    # x radius of tri wave
    global x_radius = (move_dis/wv_total_hz)
    # single wave distance
    global wave_dis = sqrt((x_radius*x_radius)+(y_radius*y_radius))*4
    # total robot distance
    global total_dis = wv_total_hz * wave_dis

    # robot speed distance/time = speed
    wv_system_speed = total_dis / (wv_times)
    if(wv_times == 0 or cir_speed_org == 0):
      write_port_register(142,111)
      sleep(0.5)
      halt
    end
    return wv_system_speed
  end


  def set_current_voltage(o_cur,o_vol):
    if(isHicomm):
      set_current_voltage_hicomm(o_cur,o_vol)
    else:
      set_current_voltage_analog(o_cur,o_vol)
    end
  end

  def set_current_voltage_hicomm(o_cur,o_vol):
      write_port_register(204,o_cur)
      write_port_register(205,o_vol*10)
      write_port_register(133,o_cur)
      write_port_register(134,o_vol*10)
  end

  def set_current_voltage_analog(o_cur,o_vol):
      vol_an=((o_vol-14)/2.8)/10
      amp_an=((o_cur-60)/44)/10
      set_standard_analog_out(0,vol_an)
      set_standard_analog_out(1,amp_an)
      write_port_register(133,o_cur)
      write_port_register(134,o_vol*10)
  end

  def calculate_2f(wving_amplitude,tg_wv_wp1,tg_wv_wp2,cir_speed_org,wving_frequency,wving_delay,wving_crater,wving_dir):
    # 진폭
    global y_radius = wving_amplitude / 2
    # 이동 거리
    global move_dis = point_dist(tg_wv_wp1,tg_wv_wp2)*1000
    global move_dis_total = move_dis
    # total running time (sec) - cir_speed_org cpm.
    global wv_times_org = move_dis/(cir_speed_org/6)
    global wv_times = wv_times_org
    global wv_total_hz = floor(wv_times_org*wving_frequency/(1+wving_delay[0]+wving_delay[1]+wving_delay[2]+wving_delay[3]))
    global get_total = wv_total_hz

    dir=1

    ratio_t_sam = 1/get_total
    T1_sam = interpolate_pose(tg_wv_wp1,tg_wv_wp2,ratio_t_sam)
    ratio_t_sam = ratio_t_sam + 1/get_total
    T2_sam = interpolate_pose(tg_wv_wp1,tg_wv_wp2,ratio_t_sam)
    ratio_t_sam = ratio_t_sam + 1/get_total
    T3_sam = interpolate_pose(tg_wv_wp1,tg_wv_wp2,ratio_t_sam)

    push_angle = wving_crater[6]
    push_dis_sam = norm(y_radius)/tan(d2r(push_angle))
    Tp1_sam = feature_offset(T2_sam,p[0,y_radius/1000,0,0,0,0],wv_Line_Feature2)
    Tp2_sam = feature_offset(T2_sam,p[0,-y_radius/1000,0,0,0,0],wv_Line_Feature2)
    Tp1_sam = feature_offset(Tp1_sam,p[wving_dir*push_dis_sam/1000,0,0,0,0,0],wv_Line_Feature2)
    Tp3_sam = feature_offset(T3_sam,p[0,-y_radius/1000,0,0,0,0],wv_Line_Feature2)
    total_step = (get_line_dist(Tp1_sam,Tp2_sam)+get_line_dist(Tp1_sam,Tp3_sam))*1000
    total_dis = wv_total_hz * total_step

    wv_system_speed = (total_dis / wv_times)

    if(wv_times == 0 or cir_speed_org == 0):
      write_port_register(142,111)
      sleep(0.5)
      halt
    end
    return wv_system_speed
  end
  def weaving_simple(wv_wp1,wv_wp3,cir_speed_org,wving_frequency,wving_amplitude,welding_on):
    wv_dist = 0
    tilt_deg = [0,0,0]
    wving_delay = [0,0,0,0]
    wving_type = 1
    Arc_sen=[0,0,0,0,0,0]
    wv_gap=[0,0,0,0]
    welding_dir=1
    z_param=[0,0,0,0,0]
    par_2f=False
    wving_crater=[0,0,0,0,0,0,0,0,0,0]
    ext_fun=[0,0,0,0,0,0,0,0,0,0,0]
    wv_seq = [0,-1]
    wv_feature=p[0,0,0,0,0,0]
    wv_weldpar=[0,cir_speed_org,0,wving_frequency,wving_amplitude,wving_type,welding_dir]
    line_weaving_tp(wv_wp1,wv_wp3,wv_weldpar,tilt_deg,wving_delay,welding_on,Arc_sen,wv_gap,z_param,par_2f,wving_crater,ext_fun,wv_seq,wv_feature)
  end

  def line_weaving_tp(wv_wp1,wv_wp3,wv_weldpar=[100,10,0,1,5,1,1,1,0],tilt_deg=[0,0,0],wving_delay=[0,0,0,0],welding_on=False,Arc_sen=[0,0,0,0,0,0],wv_gap=[0,0,0,0],z_param=[0,0,0,0,0],par_2f=False,wving_crater=[0,0,0,0,0,0,0,0,0,0],ext_fun=[0,0,0,0,0,0,0,0,0,0,0],wv_seq = [0,-1],wv_feature=p[0,0,0,0,0,0]):
    global start_gas_time = 2
    global counter_average = 1
    global counter_average_num = 0
    global waste_cycle = ext_fun[8]
    if(first_half):
      Arc_sen[1] = Arc_sen[1]/2
      Arc_sen[2] = Arc_sen[2]/2
      Arc_sen[3] = Arc_sen[3]/2
      Arc_sen[4] = Arc_sen[4]/2
    end
    global arc_x_off=0
    global arc_z_off=0
    global Up = 0
    global Ui = 0
    global Up_z = 0
    global Ui_z = 0
    if(wv_weldpar[7] == 1):
      global record_multi = False
    else:
      global record_multi = True
    end
    global th_ext_fun = ext_fun
    RTDE_init()

    # e-Series 2, CB-Seris 8
    global system_bus_ms = 2

    global sin_dir = wv_seq[1]
    global start_trig = False
    dir=1
    if(par_2f):
      global squash_cycle = 0
      # sin_dir = sin_dir
      sin_dir = sin_dir * -1
    else:
      global squash_cycle = ext_fun[7]
    end
    global tri_count=0

    global z_bottom = z_param[0]/1000
    if(wv_weldpar[6]==-1):
      #right
      global vir_v = -1
    else:
      #left
      global vir_v = 1
    end

    if(par_2f):
      global cal_off_ang_rx = 1
      global cal_off_ang_ry = 0
    else:
      global cal_off_ang_rx = 0
      global cal_off_ang_ry = 1
    end

    if(wv_seq[0] == 2 or wv_seq[0] == 3):
      tilt_deg = [0,0,0]
      global cal_off_ang_rx = 0
      global cal_off_ang_ry = 0
    end

    global wv_Line_Feature2 = wv_wp1
    if(wv_weldpar[0] > 650 and par_2f == False):
      wv_weldpar[0] = 650
    end
    if(wv_wp3==p[0,0,0,0,0,0]):
      global wv_wp2 = feature_offset(wv_wp1,p[wv_weldpar[0]/1000,0,0,0,0,0],wv_Line_Feature2)
    else:
      global wv_wp2 = wv_wp3
      wv_weldpar[0] = point_dist(wv_wp1,wv_wp2)*1000
      global wv_dist_bak = point_dist(wv_wp1,wv_wp2)*1000
    end
    if(wv_feature != p[0,0,0,0,0,0]):
      wv_Line_Feature2 = wv_feature
    end
    if(vir_v==1):
      line_x = get_feature_Line(wv_wp1,wv_wp2)
    else:
      line_x = get_feature_Line(wv_wp2,wv_wp1)
    end
    pp1 = feature_offset(wv_wp1,p[0,20/1000,0,0,0,0],line_x)
    pp2 = pose_add(wv_wp1,p[0,0,20/1000,0,0,0])
    global wp_Feature = get_feature_plane_yz(wv_wp1,pp1,pp2)

    #setting
    if(par_2f):
      #todo - 1
      global offset_2f_k = -1 * ext_fun[9]
      global offset_2f_z = 1 * ext_fun[10]
      if(wv_seq[0] == 0 or wv_seq[0] == 1):
        # line_feature = get_feature_Line(wv_wp1,wv_wp2)
        line_feature = get_feature_Line(wv_wp2,wv_wp1)
        b_p1 = wv_wp1
        b_p2 = feature_offset(wv_wp1,p[0,0.02*vir_v,0,0,0,0],line_feature)
        # b_p2 = feature_offset(wv_wp1,p[0,0.01,0,0,0,0],line_feature)
        b_p3 = pose_add(wv_wp1,p[0,0,0.02,0,0,0])

        global back_feature = get_feature_plane_xz(b_p1,b_p2,b_p3)

        wv_wp1 = pose_trans(wv_wp1,p[0,0,0,0,0,d2r(-90)])
        wv_wp1 = feature_offset(wv_wp1,p[0,offset_2f_k/1000,0,0,0,0],back_feature)
        wv_wp1 = pose_add(wv_wp1,p[0,0,offset_2f_z/1000,0,0,0])
        global bak_wv_wp1 = wv_wp1
      end
        wv_wp2 = feature_offset(wv_wp2,p[0,offset_2f_k/1000,0,0,0,0],back_feature)
        wv_wp2 = pose_add(wv_wp2,p[0,0,offset_2f_z/1000,0,0,0])
        wv_wp2 = p[wv_wp2[0],wv_wp2[1],wv_wp2[2],wv_wp1[3],wv_wp1[4],wv_wp1[5]]
        global bak_wv_wp2 = wv_wp2
    end
    if(ext_fun[2]==1 and par_2f==False):
      w_voltage = ext_fun[3]
      w_current = ext_fun[4]
      set_current_voltage(w_current,w_voltage)
      global cir_speed_org_bak = wv_weldpar[1]
      global wving_amplitude_bak = wv_weldpar[4]
      wv_weldpar[1] = ext_fun[6]
      wv_weldpar[4] = ext_fun[5]
    end
    if(par_2f):
      global wv_system_speed = calculate_2f(wv_weldpar[4],wv_wp1,wv_wp2,wv_weldpar[1],wv_weldpar[3],wving_delay,wving_crater,wv_weldpar[6])
    else:
      global wv_system_speed = calculate_3f(wv_weldpar[4],wv_wp1,wv_wp2,wv_weldpar[1],wv_weldpar[3],wving_delay)
      x_radius = x_radius / 1000
    end
    global wv_set_speed = wv_system_speed
    ratio_t=0
    global y_radius = y_radius / 1000
    global y_radius_bak = y_radius
    global ext_stick = 0
    global th_arc_sen=Arc_sen
    global th_wv_gap=wv_gap
    global th_tilt_deg=tilt_deg
    global last_tilt_deg = th_tilt_deg
    global last_wv_wp1 = wv_wp1
    global last_wv_line = wv_Line_Feature2
    global last_z_bottom = z_bottom
    global th_wving_crater=wving_crater
    global th_par_2f = par_2f
    global th_cir_speed_org=wv_weldpar[1]
    global th_wv_wp1 = wv_wp1
    global th_wv_wp2 = wv_wp2
    global th_wv_wp3 = wv_wp3
    global th_wv_weldpar=wv_weldpar
    global th_wving_delay=wving_delay
    global th_z_param=z_param
    global th_wv_seq = wv_seq
    global th_wv_feature=wv_feature
    global th_dir = dir

    # if want to use approach position
    if(wv_seq[0] ==0 or wv_seq[0] == 1):
      global get_angle_rx = welding_angle_cal_2f(wv_wp1[1],tilt_deg,vir_v,cal_off_ang_rx)
      global get_angle_ry = welding_angle_cal_3f(wv_wp1[2],tilt_deg,z_bottom,cal_off_ang_ry)

      target_p = feature_offset(wv_wp1,p[0,0,0,d2r(tilt_deg[0] + get_angle_rx),d2r(tilt_deg[1] + get_angle_ry),d2r(tilt_deg[2])],wv_Line_Feature2)

      if(wv_weldpar[2]==1):
        target_p_appr = feature_offset(target_p,p[0,0,-0.02,0,0,0],wv_Line_Feature2)
        movel(target_p_appr,a=0.5,v=0.125)
      end
      movel(target_p,a=0.5,v=0.125)
    end
    CThread = run CalThread()
    DThread = run diff_Thread()
    TThread = run thread_timer()
    AThread = run Arc_Thread()
    TTRRhread = run thread_dist_rec()

    global timer_counting=True
    global program_weld_on = True

    if(a9_wv_weldingon==True):
      while(welding_off_t==55):
        sync()
      end
      if(wving_crater[2]>0):
        set_current_voltage(wving_crater[0],wving_crater[1])
      end
      if(welding_off_t != 1):
        if(isHicomm):
          write_welder(0,True)
        else:
          set_standard_digital_out(0,True)
        end
        while(read_welder(5)==False):
          if(weld_onoff==False):
              write_welder(0,True)
          end
          sync()
        end
        if(wving_crater[2]>0):
          #Crater Begin option
          write_output_float_register(1,1)
          sleep(wving_crater[2])
          set_current_voltage(ext_fun[1],ext_fun[0])
        end
      end
    end
    start_gas_time = 0

    background_cal=1
    background_ready=0
    FT_trig=True
    timer_1_is_counting = True
    global welding_program = False

    while((ratio_t < 1)):
      if( (norm(tri_count)>=2 and par_2f==False or FT_trig==True) or (norm(tri_count)>=4 and par_2f or FT_trig==True) ):
        FT_trig = False
        while(background_ready==0):
          sync()
        end
        tri_count = 0
        background_ready = 0
        global move_p = background_pose
        wv_wp2 = th_wv_wp2
        if(par_2f):
          background_cal=1
        else:
          background_cal=1
        end
        global a_val = 3
        if(a_val >= 30):
          write_port_register(142,112)
          sleep(0.5)
          halt
        end
      end
      if(wv_weldpar[5] ==1):
          if( (sin_dir==1 and wving_delay[0]==0) or (sin_dir==-1 and wving_delay[2]==0)):
           tri_count = tri_count + 1
          end
          global target_p = move_p[tri_count]
          # write_output_float_register(24,tri_count)
          # target_p=p[target_p[0],target_p[1],target_p[2],target_p[3],target_p[4],target_p[5]]
          tri_count = tri_count + 1
      elif(wv_weldpar[5] ==2):
        if((tri_count==0 and wving_delay[2]==0) or (tri_count==2 and wving_delay[0]==0)):
         tri_count = tri_count + 1
        end
        global target_p = move_p[tri_count]
        # write_output_float_register(24,tri_count)
        # target_p=p[target_p[0],target_p[1],target_p[2],target_p[3],target_p[4],target_p[5]]
        tri_count = tri_count + 1
      else:
        popup("Please insert 0 - sin or 1 - triangle")
      end
      if(target_p == p[0,0,0,0,0,0]):
        target_p = get_actual_tcp_pose()
      end
      #3F tri_count 2 는 tri_count가 계속 move_p[1]만 간다

      # write_output_float_register(23,sin_dir)

      ARC_T_ONOFF = True
      ARC_T_s_pose = get_actual_tcp_pose()
      ARC_T_e_pose = target_p
      if((norm(tri_count)== 2) and wving_delay[1]>0 and par_2f):
        #down
        movel(target_p,a=a_val,v=wv_system_speed/1000)
        sleep(wving_delay[1])
      elif((norm(tri_count)== 4) and wving_delay[3]>0 and par_2f):
        #4
        movel(target_p,a=a_val,v=wv_system_speed/1000)
        sleep(wving_delay[3])
      elif((norm(tri_count)== 2) and sin_dir==1 and wving_delay[1]>0 and par_2f == False):
        movel(target_p,a=a_val,v=wv_system_speed/1000)
        sleep(wving_delay[1])
      elif((norm(tri_count)== 2) and sin_dir==-1 and wving_delay[3]>0 and par_2f == False):
        movel(target_p,a=a_val,v=wv_system_speed/1000)
        sleep(wving_delay[3])
      elif((norm(tri_count)== 1) and wving_delay[2]>0 and par_2f):
        movel(target_p,a=a_val,v=wv_system_speed/1000)
        sleep(wving_delay[2])
      elif((norm(tri_count)== 3) and wving_delay[0]>0 and par_2f):
        #3
        movel(target_p,a=a_val,v=wv_system_speed/1000)
        sleep(wving_delay[0])
      else:
        movel(target_p,a=a_val,v=wv_system_speed/1000)
      end
      global last_pose = target_p
    end
    timer_1_is_counting = False

    if(a9_wv_weldingon == True and wving_crater[5]!=0):
      #crater end option
      set_current_voltage(wving_crater[3],wving_crater[4])
      sleep(wving_crater[5])
      program_weld_on = False
      set_current_voltage(ext_fun[1],ext_fun[0])
      if(isHicomm):
        write_port_register(202,0)
        write_port_register(149,0)
      else:
        set_standard_digital_out(0,False)
      end
      while(read_welder(5)==True):
        if(weld_onoff==True):
          write_welder(0,False)
        end
        sync()
      end
    end
    timer_counter = 0
    kill CThread
    kill DThread
    kill TThread
    kill AThread
    kill TTRRhread
    ARC_T_ONOFF=False
    timer_counter = 0
    timer_counting = False
    wcr_counter = 0
    wcr_counting = False
    get_wcr = False
    welding_off_t = 0
    plus_alpha_x = 0
    plus_alpha_z = 0

    if(wv_seq[0] == 0 or wv_seq[0] == 3):
      if(a9_wv_weldingon==True):
        program_weld_on = False
        write_port_register(202,0)
        write_port_register(149,0)
        write_welder(0,False)
        if(wv_weldpar[2]==1):
          target_pos = feature_offset(get_actual_tcp_pose(),p[0,0,-0.01,0,0,0],wv_Line_Feature2)
          movel(target_pos,0.5,0.01)
        end
      end
    end
    background_pose = [dumy_p,dumy_p,dumy_p,dumy_p]
    move_p = background_pose
    return sin_dir
  end


  def line_weaving_tp_l(wv_wp1,wv_wp3,wv_weldpar=[100,10,0,1,5,1,1,1,0],tilt_deg=[0,0,0],wving_delay=[0,0,0,0],welding_on=False,Arc_sen=[0,0,0,0,0,0],wv_gap=[0,0,0,0],z_param=[0,0,0,0,0],par_2f=False,wving_crater=[0,0,0,0,0,0,0,0,0,0],ext_fun=[0,0,0,0,0,0,0,0,0,0,0],wv_seq = [0,-1],wv_feature=p[0,0,0,0,0,0]):
    global start_gas_time = 2
    global counter_average = 1
    global counter_average_num = 0
    global waste_cycle = ext_fun[8]
    if(first_half):
      Arc_sen[1] = Arc_sen[1]/2
      Arc_sen[2] = Arc_sen[2]/2
      Arc_sen[3] = Arc_sen[3]/2
      Arc_sen[4] = Arc_sen[4]/2
    end
    global current_list = 0
    global wv_wp4 = wv_wp3
    global A_T1 = wv_wp4[0]
    global A_T2 = wv_wp4[1]
    global A_T3 = wv_wp4[2]

    global arc_x_off=0
    global arc_z_off=0
    global Up = 0
    global Ui = 0
    global Up_z = 0
    global Ui_z = 0
    global th_ext_fun = ext_fun
    if(wv_weldpar[7] == 1):
      global record_multi = False
    else:
      global record_multi = True
    end
    RTDE_init()

    if (wv_gap[0]==1):
      gap_check = True
      wv_gap[0]=0
    else:
      gap_check= False
    end
    # e-Series 2, CB-Seris 8
    global system_bus_ms = 2

    global sin_dir = wv_seq[1]
    if(par_2f):
      global squash_cycle = 0
      # sin_dir = sin_dir
      sin_dir = sin_dir * -1
    else:
      global squash_cycle = ext_fun[7]
    end
    global start_trig = False
    dir=1

    global tri_count=0

    global z_bottom = z_param[0]/1000
    if(wv_weldpar[6]==-1):
      global vir_v = -1
    else:
      global vir_v = 1
    end

    if(par_2f):
      global cal_off_ang_rx = 1
      global cal_off_ang_ry = 0
    else:
      global cal_off_ang_rx = 0
      global cal_off_ang_ry = 1
    end

    if(wv_seq[0] == 2 or wv_seq[0] == 3):
      tilt_deg = [0,0,0]
      global cal_off_ang_rx = 0
      global cal_off_ang_ry = 0
    end

    global wv_Line_Feature2 = wv_wp1
    if(wv_weldpar[0] > 700 and par_2f == False):
      wv_weldpar[0] = 700
    end
    if(wv_wp3[0]==p[0,0,0,0,0,0]):
      global wv_wp2 = feature_offset(wv_wp1,p[wv_weldpar[0]/1000,0,0,0,0,0],wv_Line_Feature2)
    else:
      global wv_wp2 = wv_wp4[0]
      wv_weldpar[0] = point_dist(wv_wp1,wv_wp2)*1000
      global wv_dist_bak = point_dist(wv_wp1,wv_wp2)*1000
    end
    if(wv_seq[0] == 2 or wv_seq[0] == 3):
      wv_Line_Feature2 = wv_feature
    end
    if(vir_v==1):
      line_x = get_feature_Line(wv_wp1,wv_wp2)
    else:
      line_x = get_feature_Line(wv_wp2,wv_wp1)
    end  pp1 = feature_offset(wv_wp1,p[0,20/1000,0,0,0,0],line_x)
    pp2 = pose_add(wv_wp1,p[0,0,20/1000,0,0,0])
    global wp_Feature = get_feature_plane_yz(wv_wp1,pp1,pp2)

    #setting
    if(par_2f):
      #todo - 1
      offset_2f_k = -1 * ext_fun[9]
      offset_2f_z = 1 * ext_fun[10]
      if(wv_seq[0] == 0 or wv_seq[0] == 1):
        line_feature = get_feature_Line(wv_wp1,wv_wp2)
        b_p1 = wv_wp1
        b_p2 = feature_offset(wv_wp1,p[0,0.01*vir_v,0,0,0,0],line_feature)
        b_p3 = pose_add(wv_wp1,p[0,0,0.01,0,0,0])

        back_feature = get_feature_plane_xz(b_p1,b_p2,b_p3)
        wv_wp1 = pose_trans(wv_wp1,p[0,0,0,0,0,d2r(-90)])
        wv_wp1 = feature_offset(wv_wp1,p[0,offset_2f_k/1000,0,0,0,0],back_feature)
        wv_wp1 = pose_add(wv_wp1,p[0,0,offset_2f_z/1000,0,0,0])
        # wv_wp1 = pose_add(wv_wp1,p[offset_2f_k/1000,0,0,0,0,0])
      end
        # wv_wp2 = pose_add(wv_wp2,p[offset_2f_k/1000,0,0,0,0,0])
        wv_wp2 = feature_offset(wv_wp2,p[0,offset_2f_k/1000,0,0,0,0],back_feature)
        wv_wp2 = pose_add(wv_wp2,p[0,0,offset_2f_z/1000,0,0,0])
        wv_wp2 = p[wv_wp2[0],wv_wp2[1],wv_wp2[2],wv_wp1[3],wv_wp1[4],wv_wp1[5]]

        wv_wp3_p = feature_offset(wv_wp3[0],p[0,offset_2f_k/1000,0,0,0,0],back_feature)
        wv_wp3_p = pose_add(wv_wp3_p,p[0,0,offset_2f_z/1000,0,0,0])
        wv_wp3_p = p[wv_wp3_p[0],wv_wp3_p[1],wv_wp3_p[2],wv_wp1[3],wv_wp1[4],wv_wp1[5]]
        wv_wp4[0] = p[wv_wp3_p[0],wv_wp3_p[1],wv_wp3_p[2],wv_wp1[3],wv_wp1[4],wv_wp1[5]]

        wv_wp3_p = feature_offset(wv_wp3[1],p[0,offset_2f_k/1000,0,0,0,0],back_feature)
        wv_wp3_p = pose_add(wv_wp3_p,p[0,0,offset_2f_z/1000,0,0,0])
        wv_wp3_p = p[wv_wp3_p[0],wv_wp3_p[1],wv_wp3_p[2],wv_wp1[3],wv_wp1[4],wv_wp1[5]]
        wv_wp4[1] = p[wv_wp3_p[0],wv_wp3_p[1],wv_wp3_p[2],wv_wp1[3],wv_wp1[4],wv_wp1[5]]

        wv_wp3_p = feature_offset(wv_wp3[2],p[0,offset_2f_k/1000,0,0,0,0],back_feature)
        wv_wp3_p = pose_add(wv_wp3_p,p[0,0,offset_2f_z/1000,0,0,0])
        wv_wp3_p = p[wv_wp3_p[0],wv_wp3_p[1],wv_wp3_p[2],wv_wp1[3],wv_wp1[4],wv_wp1[5]]
        wv_wp4[2] = p[wv_wp3_p[0],wv_wp3_p[1],wv_wp3_p[2],wv_wp1[3],wv_wp1[4],wv_wp1[5]]
    end
    if(ext_fun[2]==1 and par_2f==False):
      #squash
      w_voltage = ext_fun[3]
      w_current = ext_fun[4]
      set_current_voltage(w_current,w_voltage)
      global cir_speed_org_bak = wv_weldpar[1]
      global wving_amplitude_bak = wv_weldpar[4]
      wv_weldpar[1] = ext_fun[6]
      wv_weldpar[4] = ext_fun[5]
    end
    if(par_2f):
      global wv_system_speed = calculate_2f(wv_weldpar[4],wv_wp1,wv_wp2,wv_weldpar[1],wv_weldpar[3],wving_delay,wving_crater,wv_weldpar[6])
    else:
      global wv_system_speed = calculate_3f(wv_weldpar[4],wv_wp1,wv_wp2,wv_weldpar[1],wv_weldpar[3],wving_delay)
      x_radius = x_radius / 1000
    end
    global wv_set_speed = wv_system_speed
    ratio_t=0
    # mm -> m
    global y_radius = y_radius / 1000
    global y_radius_bak = y_radius
    #init for thread
    global ext_stick = 0
    global th_arc_sen=Arc_sen
    global th_wv_gap=wv_gap
    global th_tilt_deg=tilt_deg

    global last_tilt_deg =th_tilt_deg
    global last_wv_wp1 = wv_wp1
    global last_wv_line = wv_Line_Feature2
    global th_wving_crater=wving_crater
    global last_z_bottom = z_bottom
    global th_par_2f = par_2f
    global th_cir_speed_org=wv_weldpar[1]
    global th_wv_wp1 = wv_wp1
    global th_wv_wp2 = wv_wp2
    global th_wv_wp3 = wv_wp3[0]
    global th_wv_weldpar=wv_weldpar
    global th_wving_delay=wving_delay
    global th_z_param=z_param
    global th_wv_seq = wv_seq
    global th_wv_feature=wv_feature
    global th_dir = dir

    # if want to use approach position
    if(wv_seq[0] ==0 or wv_seq[0] == 1):
      global get_angle_rx = welding_angle_cal_2f(wv_wp1[1],tilt_deg,vir_v,cal_off_ang_rx)
      global get_angle_ry = welding_angle_cal_3f(wv_wp1[2],tilt_deg,z_bottom,cal_off_ang_ry)

      target_p = feature_offset(wv_wp1,p[0,0,0,d2r(tilt_deg[0] + get_angle_rx),d2r(tilt_deg[1] + get_angle_ry),d2r(tilt_deg[2])],wv_Line_Feature2)

      if(wv_weldpar[2]==1):
        target_p_appr = feature_offset(target_p,p[0,0,-0.02,0,0,0],wv_Line_Feature2)
        movel(target_p_appr,a=0.5,v=0.125)
      end
      movel(target_p,a=0.5,v=0.125)
    end

    CThread = run CalThread()
    DThread = run diff_Thread()
    TThread = run thread_timer()
    AThread = run Arc_Thread()
    TTRRhread = run thread_dist_rec()

    global timer_counting=True
    global program_weld_on = True

    if(a9_wv_weldingon==True):
      while(welding_off_t==55):
        sync()
      end
      if(wving_crater[2]>0):
        set_current_voltage(wving_crater[0],wving_crater[1])
      end
      if(welding_off_t != 1):
        write_welder(0,True)
        while(get_wcr==False):
          if(weld_onoff==False):
            write_welder(0,True)
          end
          sync()
        end
        if(wving_crater[2]>0):
          #Crater Begin option
          write_output_float_register(1,1)
          sleep(wving_crater[2])
          set_current_voltage(ext_fun[1],ext_fun[0])
        end
      end
    end
    start_gas_time = 0

    background_cal=1
    background_ready=0
    FT_trig=True

    timer_1_is_counting = True

    while((ratio_t < 1) or current_list==0 or current_list==1):
      if(ratio_t>=1 and current_list!=2):
        if (gap_check):
          gap_check = True
          wv_gap[0]=1
          th_wv_gap[0]=1
          gap_check= False
        end
        ratio_t=0
        if(current_list==0):
          wving_amp_bak = wv_weldpar[4]
          wv_weldpar[4] = wv_weldpar[4] * 1
          th_wv_weldpar[4] = wv_weldpar[4]
          circle_speed_bak = wv_weldpar[1]
          wv_weldpar[1]= wv_weldpar[1]*0.7
          th_wv_weldpar[1]= wv_weldpar[1]
        elif(current_list==1):
          wv_weldpar[4] = wving_amp_bak
          th_wv_weldpar[4] = wv_weldpar[4]
          wv_weldpar[1] = circle_speed_bak
          th_wv_weldpar[1]= wv_weldpar[1]
        end
        wv_wp1=wv_wp4[current_list]
        wv_wp2=wv_wp4[current_list+1]
        global th_wv_wp1 = wv_wp4[current_list]
        global th_wv_wp2 = wv_wp4[current_list+1]
        global th_wv_wp3 = wv_wp4[current_list+1]
        wv_system_speed_bak = wv_system_speed
        if(par_2f):
          global wv_system_speed = calculate_2f(wv_weldpar[4],wv_wp4[current_list],wv_wp4[current_list+1],wv_weldpar[1],wv_weldpar[3],wving_delay,wving_crater)
          global y_radius = y_radius / 1000
          global y_radius_bak = y_radius
        else:
          global wv_system_speed = calculate_3f(wv_weldpar[4],wv_wp4[current_list],wv_wp4[current_list+1],wv_weldpar[1],wv_weldpar[3],wving_delay)
          x_radius = x_radius / 1000
        end
        wv_system_speed = wv_system_speed_bak
        current_list=current_list+1
      end

      if( (norm(tri_count)>=2 and par_2f==False or FT_trig==True) or (norm(tri_count)>=4 and par_2f==True or FT_trig==True)   ):
        FT_trig = False
        while(background_ready==0):
          sync()
        end
        tri_count = 0
        background_ready = 0
        global move_p = background_pose
        wv_wp2 = th_wv_wp2
        if(par_2f):
          background_cal=1
        else:
          background_cal=1
        end
        global a_val = 3
        if(a_val >= 30):
          write_port_register(142,112)
          sleep(0.5)
          halt
        end
      end

      if(wv_weldpar[5] ==1):
          if( (sin_dir==1 and wving_delay[0]==0) or (sin_dir==-1 and wving_delay[2]==0)):
           tri_count = tri_count + 1
          end
          # write_output_float_register(24,tri_count)
          global target_p = move_p[tri_count]
          target_p=p[target_p[0],target_p[1],target_p[2],target_p[3],target_p[4],target_p[5]]
          tri_count = tri_count + 1
      elif(wv_weldpar[5] ==2):
        if( (tri_count==1 and sin_dir==1 and wving_delay[0]==0) or (tri_count==1 and sin_dir==-1 and wving_delay[2]==0)):
         tri_count = tri_count + 1
        end
        # write_output_float_register(24,tri_count)
        global target_p = move_p[tri_count]
        target_p=p[target_p[0],target_p[1],target_p[2],target_p[3],target_p[4],target_p[5]]
        tri_count = tri_count + 1
      else:
        popup("Please insert 0 - sin or 1 - triangle")
      end

      if(target_p == p[0,0,0,0,0,0]):
        target_p = get_actual_tcp_pose()
      end
      # write_output_float_register(23,sin_dir)
      ARC_T_ONOFF = True
      ARC_T_s_pose = get_actual_tcp_pose()
      ARC_T_e_pose = target_p
      if((norm(tri_count)== 2) and wving_delay[1]>0 and par_2f):
        # DOWN
        movel(target_p,a=a_val,v=wv_system_speed/1000)
        sleep(wving_delay[1])
      elif((norm(tri_count)== 4) and wving_delay[3]>0 and par_2f):
        #UP
        movel(target_p,a=a_val,v=wv_system_speed/1000)
        sleep(wving_delay[3])
      elif((norm(tri_count)== 2) and sin_dir==1 and wving_delay[1]>0 and par_2f == False):
        movel(target_p,a=a_val,v=wv_system_speed/1000)
        sleep(wving_delay[1])
      elif((norm(tri_count)== 2) and sin_dir==-1 and wving_delay[3]>0 and par_2f == False):
        movel(target_p,a=a_val,v=wv_system_speed/1000)
        sleep(wving_delay[3])
      elif((norm(tri_count)== 1) and wving_delay[0]>0 and par_2f):
        movel(target_p,a=a_val,v=wv_system_speed/1000)
        sleep(wving_delay[0])
      elif((norm(tri_count)== 3) and wving_delay[2]>0 and par_2f):
        movel(target_p,a=a_val,v=wv_system_speed/1000)
        sleep(wving_delay[2])
      else:
        movel(target_p,a=a_val,v=wv_system_speed/1000)
      end
      global last_pose = target_p
    end

    timer_1_is_counting = False
    welding_program = True
    if(a9_wv_weldingon == True and wving_crater[5]!=0):
      #crater end option
      set_current_voltage(wving_crater[3],wving_crater[4])
      sleep(wving_crater[5])
      program_weld_on = False
      set_current_voltage(ext_fun[1],ext_fun[0])
      if(isHicomm):
        write_port_register(202,0)
        write_port_register(149,0)
      else:
        set_standard_digital_out(0,False)
      end
      while(get_wcr==True):
        if(weld_onoff==True):
          if(isHicomm):
            write_port_register(202,0)
            write_port_register(149,0)
          else:
            set_standard_digital_out(0,False)
          end
        end
        sync()
      end
    end

    kill CThread
    kill DThread
    kill TThread
    kill AThread
    kill TTRRhread
    ARC_T_ONOFF=False
    timer_counting = False
    wcr_counter = 0
    wcr_counting = False
    get_wcr = False
    welding_off_t = 0
    plus_alpha_x = 0
    plus_alpha_z = 0

    if(wv_seq[0] == 0 or wv_seq[0] == 3):
      if(a9_wv_weldingon==True):
        program_weld_on = False
        if(isHicomm):
          write_port_register(202,0)
          write_port_register(149,0)
        else:
          set_standard_digital_out(0,False)
        end
        if(wv_weldpar[2]==1):
          target_pos = feature_offset(get_actual_tcp_pose(),p[0,0,-0.01,0,0,0],wv_Line_Feature2)
          movel(target_pos,0.5,0.01)
        end
      end
    end
    background_pose = [dumy_p,dumy_p,dumy_p,dumy_p]
    move_p = background_pose
    return sin_dir
  end
  $ 152 "Reset"
  $ 153 "If Reset_Trig"
  if (Reset_Trig):
    $ 154 "Reset_Trig≔ False "
    global Reset_Trig=  False
    $ 155 "Call robotand_cell_initalizat"
    robotand_cell_initalizat()
    $ 156 "Auto_trig≔ False "
    global Auto_trig=  False
    $ 157 "write_port_register(cell_3f_2f_151,0)"
    write_port_register(cell_3f_2f_151,0)
    $ 158 "write_port_register(cell_info_152,0)"
    write_port_register(cell_info_152,0)
    $ 159 "write_port_register(weld_req_153,0)"
    write_port_register(weld_req_153,0)
    $ 160 "write_port_register(return_done_240,0)"
    write_port_register(return_done_240,0)
    $ 161 "write_port_register(robot_move_163,0)"
    write_port_register(robot_move_163,0)
    $ 162 "write_port_register(robot_pose_164,0)"
    write_port_register(robot_pose_164,0)
    $ 163 "write_port_register(182,0)"
    write_port_register(182,0)
    $ 164 "write_port_register(185,0)"
    write_port_register(185,0)
    $ 165 "write_port_register(201,0)"
    write_port_register(201,0)
    $ 166 "write_port_register(202,0)"
    write_port_register(202,0)
  end
  $ 167 "Welding_Init"
  $ 168 "'welding parameter initialization'"
  # 'welding parameter initialization'
  $ 169 "welding_etc"
  $ 197 "c5_wv_gap_y≔0"
  global c5_wv_gap_y=0
  $ 198 "c6_wv_gap_cpm≔0"
  global c6_wv_gap_cpm=0
  $ 199 "c9_wv_gap_freq≔0"
  global c9_wv_gap_freq=0
  $ 200 "c4_gap_enable≔0"
  global c4_gap_enable=0
  $ 201 "c7_wv_gap≔[c4_gap_enable,c5_wv_gap_y,c6_wv_gap_cpm,c9_wv_gap_freq]"
  global c7_wv_gap=[c4_gap_enable,c5_wv_gap_y,c6_wv_gap_cpm,c9_wv_gap_freq]
  $ 202 "init_reset_modbus_server"
  $ 203 "set_tool_voltage(24)"
  set_tool_voltage(24)
  $ 204 "write_port_register(163,0)"
  write_port_register(163,0)
  $ 205 "write_port_register(164,0)"
  write_port_register(164,0)
  $ 207 "write_port_register(201,1)"
  write_port_register(201,1)
  $ 208 "write_port_register(202,0)"
  write_port_register(202,0)
  $ 1310 "Thread_2"
  thread Thread_2():
    while (True):
      $ 1311 "Thread_heartbeat"
      $ 1312 "heartbeat≔heartbeat+1"
      global heartbeat=heartbeat+1
      $ 1313 "If heartbeat>499"
      if (heartbeat>499):
        $ 1314 "heartbeat≔0"
        global heartbeat=0
      end
      $ 1315 "write_port_register(128,heartbeat)"
      write_port_register(128,heartbeat)
      $ 1325 "Wait: 1.0"
      sleep(1.0)
    end
  end
  threadId_Thread_2 = run Thread_2()
  $ 1326 "Thread_1"
  thread Thread_1():
    while (True):
      $ 1327 "thread main"
      $ 1328 "a0_Job_Mode≔read_port_register(162)"
      global a0_Job_Mode= read_port_register (162)
      $ 1329 "a1_job_move≔read_port_register(163)"
      global a1_job_move= read_port_register (163)
      $ 1330 "If red_led≟ True "
      if (get_tool_digital_out(0) ==   True  ):
        $ 1331 "Set red_led=Off"
        set_tool_digital_out(0, False)
      end
      $ 1332 "If a0_Job_Mode≟2"
      if (a0_Job_Mode == 2):
        $ 1333 "If read_port_register(arc_onoff_168)≟2"
        if ( read_port_register (arc_onoff_168) == 2):
          $ 1334 "a9_wv_weldingon≔ True "
          global a9_wv_weldingon=  True
        else:
          $ 1335 "Else" "noBreak"
          $ 1336 "a9_wv_weldingon≔ False "
          global a9_wv_weldingon=  False
        end
        $ 1337 "If Auto_trig"
        if (Auto_trig):
          $ 1338 "get_next_number≔read_port_register(166)"
          global get_next_number= read_port_register (166)
          $ 1339 "get_move_trig≔read_port_register(167)"
          global get_move_trig= read_port_register (167)
          $ 1340 "If get_move_trig≟1 and running_trig≟ True "
          if (get_move_trig == 1  and  running_trig ==   True  ):
            $ 1341 "If get_next_number<0 or get_next_number>30"
            if (get_next_number<0  or  get_next_number>30):
              $ 1342 "write_port_register(142,141)"
              write_port_register(142,141)
              $ 1343 "Halt"
              halt
            end
            $ 1344 "If get_next_number≠Auto_cur_cell"
            if (get_next_number != Auto_cur_cell):
              $ 1345 "running_trig≔ False "
              global running_trig=  False
              $ 1346 "write_welder(0, False )"
              write_welder(0,  False  )
              $ 1347 "write_port_register(149,0)"
              write_port_register(149,0)
              $ 1348 "write_port_register(202,0)"
              write_port_register(202,0)
            else:
              $ 1349 "Else" "noBreak"
              $ 1350 "write_port_register(166,0)"
              write_port_register(166,0)
              $ 1351 "write_port_register(167,0)"
              write_port_register(167,0)
            end
          end
        end
        $ 1352 "If t_time>timer_1"
        if (t_time>timer_1):
          $ 1353 "write_port_register(143,timer_1)"
          write_port_register(143,timer_1)
        else:
          $ 1354 "Else" "noBreak"
          $ 1355 "write_port_register(143,timer_1)"
          write_port_register(143,timer_1)
          $ 1356 "write_port_register(144,timer_1)"
          write_port_register(144,timer_1)
        end
        $ 1357 "Monitoring touch and welding"
        $ 1358 "If read_welder_control(0) and read_port_register(130)≠1"
        if (read_welder_control(0)  and   read_port_register (130) != 1):
          $ 1359 "write_port_register(130,1)"
          write_port_register(130,1)
        else:
          $ 1360 "ElseIf read_welder_control(0) and read_port_register(130)≠0"
          if (read_welder_control(0)  and   read_port_register (130) != 0):
            $ 1361 "write_port_register(130,0)"
            write_port_register(130,0)
          end
        end
        $ 1362 "If read_welder(5)"
        if (read_welder(5)):
          $ 1363 "'check wcr in (digital)'"
          # 'check wcr in (digital)'
          $ 1364 "write_output_float_register(20,1)"
          write_output_float_register(20,1)
        else:
          $ 1365 "Else" "noBreak"
          $ 1366 "write_output_float_register(20,0)"
          write_output_float_register(20,0)
        end
        $ 1367 "If read_welder(4)"
        if (read_welder(4)):
          $ 1368 "'check touch (digital)'"
          # 'check touch (digital)'
          $ 1369 "write_output_float_register(21,1)"
          write_output_float_register(21,1)
        else:
          $ 1370 "Else" "noBreak"
          $ 1371 "write_output_float_register(21,0)"
          write_output_float_register(21,0)
        end
        $ 1372 "If read_welder_control(0)"
        if (read_welder_control(0)):
          $ 1373 "'check welding out (digital)'"
          # 'check welding out (digital)'
          $ 1374 "write_output_float_register(17,1)"
          write_output_float_register(17,1)
        else:
          $ 1375 "Else" "noBreak"
          $ 1376 "write_output_float_register(17,0)"
          write_output_float_register(17,0)
        end
        $ 1377 "If read_welder_control(4)"
        if (read_welder_control(4)):
          $ 1378 "'check touch out (digital)'"
          # 'check touch out (digital)'
          $ 1379 "write_output_float_register(18,1)"
          write_output_float_register(18,1)
        else:
          $ 1380 "Else" "noBreak"
          $ 1381 "write_output_float_register(18,0)"
          write_output_float_register(18,0)
        end
      end
      $ 1382 "If get_tool_digital_in(1)≟ True "
      if (get_tool_digital_in(1) ==   True  ):
        $ 1383 "set_tool_digital_out(1, False )"
        set_tool_digital_out(1,  False  )
      else:
        $ 1384 "Else" "noBreak"
        $ 1385 "set_tool_digital_out(1, True )"
        set_tool_digital_out(1,  True  )
      end
      $ 1386 "If red_led≟ True "
      if (get_tool_digital_out(0) ==   True  ):
        $ 1387 "Set red_led=Off"
        set_tool_digital_out(0, False)
        $ 1388 "end_freedrive_mode()"
        end_freedrive_mode()
      end
      $ 1389 "check_speed()"
      check_speed()
      $ 1390 "Wait: 0.05"
      sleep(0.05)
    end
  end
  threadId_Thread_1 = run Thread_1()
  thread EventThread():
    while (True):
      if (event_cal_on):
        $ 1392 "calculate_position"
        $ 1395 "move_i_f≔1"
        global move_i_f=1
        $ 1396 "get_pose_side≔0"
        global get_pose_side=0
        $ 1397 "Loop move_i_f<10"
        while (move_i_f<10):
          $ 1398 "If A_Touch_trig_l[move_i_f]≟ True "
          if (A_Touch_trig_l[move_i_f] ==   True  ):
            $ 1399 "If move_i_f≟A_VL1 or move_i_f≟A_VL2"
            if (move_i_f == A_VL1  or  move_i_f == A_VL2):
              $ 1400 "A_sel_v≔move_i_f"
              global A_sel_v=move_i_f
              $ 1401 "If simulation_mode"
              if (simulation_mode):
                $ 1402 "Call welding_parameter_sim"
                welding_parameter_sim()
              else:
                $ 1403 "Else" "noBreak"
                $ 1404 "Call welding_parameter_init"
                welding_parameter_init()
              end
              $ 1405 "If a8_wv_distance<5"
              if (a8_wv_distance<5):
                $ 1406 "write_port_register(142,143)"
                write_port_register(142,143)
                $ 1407 "Halt"
                halt
              end
              $ 1408 "b2_left_par≔ True "
              global b2_left_par=  True
              $ 1409 "b8_wv_2f≔ False "
              global b8_wv_2f=  False
              $ 1410 "If move_i_f≟A_VL2"
              if (move_i_f == A_VL2):
                $ 1411 "callar_hor≔a6_callar_hor"
                global callar_hor=a6_callar_hor
                $ 1412 "If b1_cell_info_L≟E or b1_cell_info_L≟e"
                if (b1_cell_info_L == E  or  b1_cell_info_L == e):
                  $ 1413 "'For bottom touch(zero) after offset not used now'"
                  # 'For bottom touch(zero) after offset not used now'
                  $ 1414 "vert_scallup_l≔a5_f_hole[1]"
                  global vert_scallup_l=a5_f_hole[1]
                end
                $ 1415 "b2_cell≔b1_cell_info_L"
                global b2_cell=b1_cell_info_L
                $ 1416 "get_pos≔get_lr(up_left,a6_f_width,a5_f_hole,a7_f_distance,b2_left_par,b8_wv_2f,Touch_dis,get_margin_z,touch_side,callar_hor,b2_cell,center_line)"
                global get_pos=get_lr(p[.492775857339, .409517380626, -.029063830209, -2.419264859926, -.998084331190, -1.368689080860],a6_f_width,a5_f_hole,a7_f_distance,b2_left_par,b8_wv_2f,Touch_dis,get_margin_z,touch_side,callar_hor,b2_cell,center_line)
              else:
                $ 1419 "Else" "noBreak"
                $ 1420 "callar_hor≔0"
                global callar_hor=0
                $ 1421 "'For bottom touch(zero) after offset not used now'"
                # 'For bottom touch(zero) after offset not used now'
                $ 1422 "vert_scallup_l≔a5_f_hole[1]"
                global vert_scallup_l=a5_f_hole[1]
                $ 1423 "b2_cell≔b1_cell_info_L"
                global b2_cell=b1_cell_info_L
                $ 1424 "get_pos≔get_lr(left,a6_f_width,a5_f_hole,a7_f_distance,b2_left_par,b8_wv_2f,Touch_dis,get_margin_z,touch_side,callar_hor,b2_cell,center_line)"
                global get_pos=get_lr(p[.480496318984, .411279115151, .006998291210, -2.211681476386, -.899147924387, -1.383032568605],a6_f_width,a5_f_hole,a7_f_distance,b2_left_par,b8_wv_2f,Touch_dis,get_margin_z,touch_side,callar_hor,b2_cell,center_line)
              end
              $ 1425 "pre_tp≔tilt_3f_fun(get_pos,[0,0,0],0)"
              global pre_tp=tilt_3f_fun(get_pos,[0,0,0],0)
              $ 1426 "A_Prepos_l[move_i_f]=pre_tp"
              A_Prepos_l[move_i_f]=pre_tp
            else:
              $ 1427 "ElseIf move_i_f≟A_VR1 or move_i_f≟A_VR2"
              if (move_i_f == A_VR1  or  move_i_f == A_VR2):
                $ 1428 "A_sel_v≔move_i_f"
                global A_sel_v=move_i_f
                $ 1429 "If simulation_mode"
                if (simulation_mode):
                  $ 1430 "Call welding_parameter_sim"
                  welding_parameter_sim()
                else:
                  $ 1431 "Else" "noBreak"
                  $ 1432 "Call welding_parameter_init"
                  welding_parameter_init()
                end
                $ 1433 "If a8_wv_distance<5"
                if (a8_wv_distance<5):
                  $ 1434 "write_port_register(142,143)"
                  write_port_register(142,143)
                  $ 1435 "Halt"
                  halt
                end
                $ 1436 "b2_left_par≔ False "
                global b2_left_par=  False
                $ 1437 "b8_wv_2f≔ False "
                global b8_wv_2f=  False
                $ 1438 "If move_i_f≟A_VR2"
                if (move_i_f == A_VR2):
                  $ 1439 "callar_hor≔a6_callar_hor"
                  global callar_hor=a6_callar_hor
                  $ 1440 "If b1_cell_info_R≟E or b1_cell_info_R≟e"
                  if (b1_cell_info_R == E  or  b1_cell_info_R == e):
                    $ 1441 "vert_scallup_r≔a5_f_hole[1]"
                    global vert_scallup_r=a5_f_hole[1]
                  end
                  $ 1442 "b2_cell≔b1_cell_info_R"
                  global b2_cell=b1_cell_info_R
                  $ 1443 "get_pos≔get_lr(up_right,a6_f_width,a5_f_hole,a7_f_distance,b2_left_par,b8_wv_2f,Touch_dis,get_margin_z,touch_side,callar_hor,b2_cell,center_line)"
                  global get_pos=get_lr(p[.445203173045, -.406687378356, -.031125942276, 2.308490741423, -1.066468937023, 1.322151316133],a6_f_width,a5_f_hole,a7_f_distance,b2_left_par,b8_wv_2f,Touch_dis,get_margin_z,touch_side,callar_hor,b2_cell,center_line)
                else:
                  $ 1446 "Else" "noBreak"
                  $ 1447 "callar_hor≔0"
                  global callar_hor=0
                  $ 1448 "vert_scallup_r≔a5_f_hole[1]"
                  global vert_scallup_r=a5_f_hole[1]
                  $ 1449 "b2_cell≔b1_cell_info_R"
                  global b2_cell=b1_cell_info_R
                  $ 1450 "get_pos≔get_lr(right,a6_f_width,a5_f_hole,a7_f_distance,b2_left_par,b8_wv_2f,Touch_dis,get_margin_z,touch_side,callar_hor,b2_cell,center_line)"
                  global get_pos=get_lr(p[.475000000000, -.421403215678, .026417194146, 1.917761036827, -1.141682393512, 1.523356199292],a6_f_width,a5_f_hole,a7_f_distance,b2_left_par,b8_wv_2f,Touch_dis,get_margin_z,touch_side,callar_hor,b2_cell,center_line)
                end
                $ 1451 "pre_tp≔tilt_3f_fun(get_pos,[0,0,0],0)"
                global pre_tp=tilt_3f_fun(get_pos,[0,0,0],0)
                $ 1452 "A_Prepos_l[move_i_f]=pre_tp"
                A_Prepos_l[move_i_f]=pre_tp
              else:
                $ 1453 "ElseIf move_i_f≟A_HOR"
                if (move_i_f == A_HOR):
                  $ 1454 "A_sel_v≔A_HOR"
                  global A_sel_v=A_HOR
                  $ 1455 "If simulation_mode"
                  if (simulation_mode):
                    $ 1456 "Call welding_parameter_sim"
                    welding_parameter_sim()
                  else:
                    $ 1457 "Else" "noBreak"
                    $ 1458 "Call welding_parameter_init"
                    welding_parameter_init()
                  end
                  $ 1459 "hor_l_scallup≔a5_f_hole[1]"
                  global hor_l_scallup=a5_f_hole[1]
                  $ 1460 "b8_wv_2f≔ True "
                  global b8_wv_2f=  True
                  $ 1461 "b2_left_par≔ True "
                  global b2_left_par=  True
                  $ 1462 "b2_cell≔b1_cell_info_L"
                  global b2_cell=b1_cell_info_L
                  $ 1463 "get_pos≔get_lr(up_left,a6_f_width,a5_f_hole,a7_f_distance,b2_left_par,b8_wv_2f,Touch_dis,get_margin_z,touch_side,0,b2_cell,center_line)"
                  global get_pos=get_lr(p[.492775857339, .409517380626, -.029063830209, -2.419264859926, -.998084331190, -1.368689080860],a6_f_width,a5_f_hole,a7_f_distance,b2_left_par,b8_wv_2f,Touch_dis,get_margin_z,touch_side,0,b2_cell,center_line)
                  $ 1464 "pre_tp≔get_pos"
                  global pre_tp=get_pos
                  $ 1465 "A_Prepos_l[move_i_f]=pre_tp"
                  A_Prepos_l[move_i_f]=pre_tp
                else:
                  $ 1466 "ElseIf move_i_f≟A_HOR_R"
                  if (move_i_f == A_HOR_R):
                    $ 1467 "A_sel_v≔A_HOR"
                    global A_sel_v=A_HOR
                    $ 1468 "If simulation_mode"
                    if (simulation_mode):
                      $ 1469 "Call welding_parameter_sim"
                      welding_parameter_sim()
                    else:
                      $ 1470 "Else" "noBreak"
                      $ 1471 "Call welding_parameter_init"
                      welding_parameter_init()
                    end
                    $ 1472 "hor_r_scallup≔a5_f_hole[2]"
                    global hor_r_scallup=a5_f_hole[2]
                    $ 1473 "b2_left_par≔ False "
                    global b2_left_par=  False
                    $ 1474 "b8_wv_2f≔ True "
                    global b8_wv_2f=  True
                    $ 1475 "b2_cell≔b1_cell_info_R"
                    global b2_cell=b1_cell_info_R
                    $ 1476 "get_pos≔get_lr(up_right,a6_f_width,a5_f_hole,a7_f_distance,b2_left_par,b8_wv_2f,Touch_dis,get_margin_z,touch_side,0,b2_cell,center_line)"
                    global get_pos=get_lr(p[.445203173045, -.406687378356, -.031125942276, 2.308490741423, -1.066468937023, 1.322151316133],a6_f_width,a5_f_hole,a7_f_distance,b2_left_par,b8_wv_2f,Touch_dis,get_margin_z,touch_side,0,b2_cell,center_line)
                    $ 1477 "pre_tp≔get_pos"
                    global pre_tp=get_pos
                    $ 1478 "A_Prepos_l[move_i_f]=pre_tp"
                    A_Prepos_l[move_i_f]=pre_tp
                  else:
                    $ 1479 "ElseIf move_i_f≟A_HOR_ML"
                    if (move_i_f == A_HOR_ML):
                      $ 1480 "A_sel_v≔A_HOR_ML"
                      global A_sel_v=A_HOR_ML
                      $ 1481 "If simulation_mode"
                      if (simulation_mode):
                        $ 1482 "Call welding_parameter_sim"
                        welding_parameter_sim()
                      else:
                        $ 1483 "Else" "noBreak"
                        $ 1484 "Call welding_parameter_init"
                        welding_parameter_init()
                      end
                      $ 1485 "b8_wv_2f≔ True "
                      global b8_wv_2f=  True
                      $ 1486 "b2_left_par≔ True "
                      global b2_left_par=  True
                      $ 1487 "b2_cell≔b1_cell_info_L"
                      global b2_cell=b1_cell_info_L
                      $ 1488 "Touch_dis≔-1*Touch_dis"
                      global Touch_dis=-1*Touch_dis
                      $ 1489 "get_pos≔get_lr(up_left,a6_f_width,a5_f_hole,a7_f_distance,b2_left_par,b8_wv_2f,Touch_dis,get_margin_z,touch_side,a6_callar_hor,b2_cell,center_line)"
                      global get_pos=get_lr(p[.492775857339, .409517380626, -.029063830209, -2.419264859926, -.998084331190, -1.368689080860],a6_f_width,a5_f_hole,a7_f_distance,b2_left_par,b8_wv_2f,Touch_dis,get_margin_z,touch_side,a6_callar_hor,b2_cell,center_line)
                      $ 1490 "Touch_dis≔-1*Touch_dis"
                      global Touch_dis=-1*Touch_dis
                      $ 1491 "pre_tp≔get_pos"
                      global pre_tp=get_pos
                      $ 1492 "A_Prepos_l[move_i_f]=pre_tp"
                      A_Prepos_l[move_i_f]=pre_tp
                    else:
                      $ 1493 "ElseIf move_i_f≟A_HOR_MR"
                      if (move_i_f == A_HOR_MR):
                        $ 1494 "A_sel_v≔A_HOR_MR"
                        global A_sel_v=A_HOR_MR
                        $ 1495 "If simulation_mode"
                        if (simulation_mode):
                          $ 1496 "Call welding_parameter_sim"
                          welding_parameter_sim()
                        else:
                          $ 1497 "Else" "noBreak"
                          $ 1498 "Call welding_parameter_init"
                          welding_parameter_init()
                        end
                        $ 1499 "b2_left_par≔ False "
                        global b2_left_par=  False
                        $ 1500 "b8_wv_2f≔ True "
                        global b8_wv_2f=  True
                        $ 1501 "b2_cell≔b1_cell_info_R"
                        global b2_cell=b1_cell_info_R
                        $ 1502 "Touch_dis≔-1*Touch_dis"
                        global Touch_dis=-1*Touch_dis
                        $ 1503 "get_pos≔get_lr(up_right,a6_f_width,a5_f_hole,a7_f_distance,b2_left_par,b8_wv_2f,Touch_dis,get_margin_z,touch_side,a6_callar_hor,b2_cell,center_line)"
                        global get_pos=get_lr(p[.445203173045, -.406687378356, -.031125942276, 2.308490741423, -1.066468937023, 1.322151316133],a6_f_width,a5_f_hole,a7_f_distance,b2_left_par,b8_wv_2f,Touch_dis,get_margin_z,touch_side,a6_callar_hor,b2_cell,center_line)
                        $ 1504 "Touch_dis≔-1*Touch_dis"
                        global Touch_dis=-1*Touch_dis
                        $ 1505 "pre_tp≔get_pos"
                        global pre_tp=get_pos
                        $ 1506 "A_Prepos_l[move_i_f]=pre_tp"
                        A_Prepos_l[move_i_f]=pre_tp
                      end
                    end
                  end
                end
              end
            end
            $ 1507 "If move_i_f≤4"
            if (move_i_f <= 4):
              $ 1508 "A_Prepos_l[move_i_f+9]=p[0,0,0,0,0,0]"
              A_Prepos_l[move_i_f+9]=p[0,0,0,0,0,0]
            end
          end
          $ 1511 "move_i_f≔move_i_f+1"
          global move_i_f=move_i_f+1
        end
        $ 1512 "event_cal_on≔ False "
        global event_cal_on=  False
      elif (event_side_on):
        $ 1514 "calculate_side"
        $ 1517 "Wait event_cal_on≟ False "
        while (not(event_cal_on ==   False  )):
          sync()
        end
        $ 1518 "move_i_f≔1"
        global move_i_f=1
        $ 1519 "get_pose_side≔get_pose_side_t"
        global get_pose_side=get_pose_side_t
        $ 1520 "Loop move_i_f<10"
        while (move_i_f<10):
          $ 1521 "If A_Touch_trig_l[move_i_f]≟ True "
          if (A_Touch_trig_l[move_i_f] ==   True  ):
            $ 1522 "If move_i_f≟A_VL1 or move_i_f≟A_VL2"
            if (move_i_f == A_VL1  or  move_i_f == A_VL2):
              $ 1523 "A_Prepos_l[move_i_f]=side_apply(A_Prepos_l[move_i_f],center_line,get_pose_side)"
              A_Prepos_l[move_i_f]=side_apply(A_Prepos_l[move_i_f],center_line,get_pose_side)
            else:
              $ 1524 "ElseIf move_i_f≟A_VR1 or move_i_f≟A_VR2"
              if (move_i_f == A_VR1  or  move_i_f == A_VR2):
                $ 1525 "A_Prepos_l[move_i_f]=side_apply(A_Prepos_l[move_i_f],center_line,get_pose_side)"
                A_Prepos_l[move_i_f]=side_apply(A_Prepos_l[move_i_f],center_line,get_pose_side)
              else:
                $ 1526 "ElseIf move_i_f≟A_HOR"
                if (move_i_f == A_HOR):
                  $ 1527 "A_Prepos_l[move_i_f]=side_apply(A_Prepos_l[move_i_f],center_line,get_pose_side)"
                  A_Prepos_l[move_i_f]=side_apply(A_Prepos_l[move_i_f],center_line,get_pose_side)
                else:
                  $ 1528 "ElseIf move_i_f≟A_HOR_R"
                  if (move_i_f == A_HOR_R):
                    $ 1529 "A_Prepos_l[move_i_f]=side_apply(A_Prepos_l[move_i_f],center_line,get_pose_side)"
                    A_Prepos_l[move_i_f]=side_apply(A_Prepos_l[move_i_f],center_line,get_pose_side)
                  else:
                    $ 1530 "ElseIf move_i_f≟A_HOR_ML"
                    if (move_i_f == A_HOR_ML):
                      $ 1531 "A_Prepos_l[move_i_f]=side_apply(A_Prepos_l[move_i_f],center_line,get_pose_side)"
                      A_Prepos_l[move_i_f]=side_apply(A_Prepos_l[move_i_f],center_line,get_pose_side)
                    else:
                      $ 1532 "ElseIf move_i_f≟A_HOR_MR"
                      if (move_i_f == A_HOR_MR):
                        $ 1533 "A_Prepos_l[move_i_f]=side_apply(A_Prepos_l[move_i_f],center_line,get_pose_side)"
                        A_Prepos_l[move_i_f]=side_apply(A_Prepos_l[move_i_f],center_line,get_pose_side)
                      end
                    end
                  end
                end
              end
            end
          end
          $ 1534 "move_i_f≔move_i_f+1"
          global move_i_f=move_i_f+1
        end
        $ 1535 "event_side_on≔ False "
        global event_side_on=  False
      elif (reset_trig):
        $ 1537 "Call reset_weld_param"
        reset_weld_param()
        $ 1538 "reset_trig≔ False "
        global reset_trig=  False
      elif (time_cal_trig):
        $ 1540 "t_time≔time_cal(Auto_W_num,Auto_total_cell,A_Speed_list,A_Distance_list,A_Touch_p,0)"
        global t_time=time_cal(Auto_W_num,Auto_total_cell,A_Speed_list,A_Distance_list,A_Touch_p,0)
        $ 1541 "write_port_register(144,t_time)"
        write_port_register(144,t_time)
        $ 1542 "time_cal_trig≔ False "
        global time_cal_trig=  False
      elif (pause_trig):
        $ 1544 "s_conn≔socket_open('192.168.1.7',29999)"
        global s_conn=socket_open("192.168.1.7",29999)
        $ 1545 "s_send≔socket_send_string('pause')"
        global s_send=socket_send_string("pause")
        $ 1546 "s_send≔socket_send_byte(10)"
        global s_send=socket_send_byte(10)
        $ 1547 "socket_close()"
        socket_close()
        $ 1548 "pause_trig≔ False "
        global pause_trig=  False
      end
      sync()
    end
  end
  eventThread = run EventThread()
  while (True):
    $ 209 "Robot Program"
    $ 227 "If simulation_mode"
    if (simulation_mode):
      $ 228 "'work mode 2'"
      # 'work mode 2'
      $ 229 "write_port_register(162,2)"
      write_port_register(162,2)
      $ 230 "touch_temp≔0"
      global touch_temp=0
    end
    $ 231 "If a0_Job_Mode≟1"
    if (a0_Job_Mode == 1):
      $ 232 "job mode 1"
      $ 233 "'JOB_MANUAL'"
      # 'JOB_MANUAL'
      $ 234 "write_port_register(robot_ready_141,1)"
      write_port_register(robot_ready_141,1)
      $ 235 "If freedrive≟ True  and freedrive_trg≟ False "
      if (get_tool_digital_in(1) ==   True    and  freedrive_trg ==   False  ):
        $ 236 "freedrive_trg≔ True "
        global freedrive_trg=  True
        $ 237 "freedrive_mode()"
        freedrive_mode()
      else:
        $ 238 "ElseIf freedrive≟ False  and freedrive_trg≟ True "
        if (get_tool_digital_in(1) ==   False    and  freedrive_trg ==   True  ):
          $ 239 "end_freedrive_mode()"
          end_freedrive_mode()
          $ 240 "freedrive_trg≔ False "
          global freedrive_trg=  False
        end
      end
      $ 244 "If freedrive≟ True  and save_tool≟ True "
      if (get_tool_digital_in(1) ==   True    and  get_tool_digital_in(0) ==   True  ):
        $ 248 "Wait: 0.01"
        sleep(0.01)
      else:
        $ 249 "ElseIf a1_job_move≟1"
        if (a1_job_move == 1):
          $ 250 "'Manual - Move Home/Packing/Warmup'"
          # 'Manual - Move Home/Packing/Warmup'
          $ 251 "If read_port_register(robot_pose_164)≟1"
          if ( read_port_register (robot_pose_164) == 1):
            $ 252 "write_port_register(robot_ready_141,0)"
            write_port_register(robot_ready_141,0)
            $ 253 "homeing()"
            homeing()
            $ 254 "MoveJ"
            $ 255 "Packing_pos" "breakAfter"
            movej([1.5877798795700073, -0.0173419157611292, -2.4983108679400843, -1.4065726439105433, 1.626846194267273, 3.0169763565063477], a=0.9599310885968813, v=0.9599310885968813)
          else:
            $ 256 "ElseIf read_port_register(robot_pose_164)≟2"
            if ( read_port_register (robot_pose_164) == 2):
              $ 257 "write_port_register(robot_ready_141,0)"
              write_port_register(robot_ready_141,0)
              $ 258 "homeing()"
              homeing()
            else:
              $ 259 "ElseIf read_port_register(robot_pose_164)≟3"
              global thread_flag_259=0
              thread Thread_if_259():
                $ 260 "write_port_register(robot_ready_141,0)"
                write_port_register(robot_ready_141,0)
                $ 261 "Warm-up"
                $ 262 "Loop 22 times"
                Loop_9 = 0
                while (Loop_9 < 22):
                  $ 263 "MoveJ"
                  $ 264 "Warming_1" "breakAfter"
                  movej([1.0598392486572266, -1.0896032492267054, -1.2158034483539026, -2.3403762022601526, 1.497584342956543, 2.354665517807007], a=0.17453292519943295, v=0.08726646259971647)
                  $ 265 "Warming_2" "breakAfter"
                  movej([0.7106529474258423, -1.0894954840289515, -1.215731445943014, -2.3402441183673304, 1.4977161884307861, 2.3545455932617188], a=0.17453292519943295, v=0.08726646259971647)
                  $ 266 "Warming_3" "breakAfter"
                  movej([0.8852421641349792, -1.0894234816180628, -1.215863052998678, -2.340435806904928, 1.497644305229187, 2.3545212745666504], a=0.17453292519943295, v=0.08726646259971647)
                  $ 267 "Warming_4" "breakAfter"
                  movej([0.885266125202179, -1.263935391102926, -1.2099388281451624, -2.352635685597555, 1.4888625144958496, 2.3787333965301514], a=0.17453292519943295, v=0.08726646259971647)
                  $ 268 "Wariming_5" "breakAfter"
                  movej([0.8852541446685791, -0.9149578253375452, -1.217938248311178, -2.335618321095602, 1.501125693321228, 2.3452301025390625], a=0.17453292519943295, v=0.08726646259971647)
                  $ 269 "Warming_6" "breakAfter"
                  movej([0.8852177858352661, -1.0895074049579065, -1.3828147093402308, -2.343850914631979, 1.489568829536438, 2.3598153591156006], a=0.17453292519943295, v=0.08726646259971647)
                  $ 270 "Warming_7" "breakAfter"
                  movej([0.885229766368866, -1.0894115606891077, -1.220372502003805, -2.335630242024557, 1.5009583234786987, 2.3453502655029297], a=0.17453292519943295, v=0.08726646259971647)
                  $ 271 "Warming_8" "breakAfter"
                  movej([0.6920775233962951, -1.0506328608604214, -1.2152130579572011, -2.5072867131215766, 1.4917910996963177, 2.3459413556024855], a=0.17453292519943295, v=0.08726646259971647)
                  $ 272 "Warming_9" "breakAfter"
                  movej([0.6929177641868591, -1.0475013891803187, -1.2503178755389612, -2.327541176472799, 1.5014369487762451, 2.345398187637329], a=0.17453292519943295, v=0.08726646259971647)
                  $ 273 "Warming_10" "breakAfter"
                  movej([0.8162043690681458, -1.1462538878070276, -1.3285825888263147, -2.3897975126849573, 1.2906681299209595, 2.3704988956451416], a=0.17453292519943295, v=0.08726646259971647)
                  $ 274 "Warming_11" "breakAfter"
                  movej([0.6952417412291937, -1.0226626805382075, -1.3187663864026051, -2.3852732107244847, 1.5281305955128988, 2.3484138521676003], a=0.17453292519943295, v=0.08726646259971647)
                  $ 275 "Warming_12" "breakAfter"
                  movej([0.6938896179199219, -1.0222962538348597, -1.3204510847674769, -2.403698269520895, 1.7271294593811035, 2.3448219299316406], a=0.17453292519943295, v=0.08726646259971647)
                  $ 276 "Warming_13" "breakAfter"
                  movej([0.685538113117218, -1.038980786000387, -1.3163254896747034, -2.3712590376483362, 1.5282130241394043, 2.0345256328582764], a=0.17453292519943295, v=0.08726646259971647)
                  $ 277 "Warming_14" "breakAfter"
                  movej([0.721284806728363, -1.0075753370868128, -1.3205111662494105, -2.399587933217184, 1.5282011032104492, 2.539506673812866], a=0.17453292519943295, v=0.08726646259971647)
                  Loop_9 = Loop_9 + 1
                end
                $ 278 "homeing()"
                homeing()
                $ 279 "Wait: 2.0"
                sleep(2.0)
                thread_flag_259 = 1
              end
              if ( read_port_register (robot_pose_164) == 3):
                global thread_handler_259=run Thread_if_259()
                while (thread_flag_259 == 0):
                  if not( read_port_register (robot_pose_164) == 3):
                    kill thread_handler_259
                    thread_flag_259 = 2
                  else:
                    sync()
                  end
                end
              else:
                thread_flag_259 = 2
              end
              if (thread_flag_259 == 2):
                $ 280 "ElseIf read_port_register(robot_pose_164)≟4"
                if ( read_port_register (robot_pose_164) == 4):
                  $ 281 "write_port_register(robot_ready_141,0)"
                  write_port_register(robot_ready_141,0)
                  $ 282 "homeing()"
                  homeing()
                  $ 283 "MoveJ"
                  $ 284 "pre_mounting" "breakAfter"
                  movej([1.2356762886047363, -0.8703244368182581, -0.942230526600973, -2.3905327955829065, 1.3216267824172974, 2.6514604091644287], a=0.7853981633974483, v=0.7853981633974483)
                  $ 285 "Mounting_pos" "breakAfter"
                  movej([0.6231353085164267, -0.6300961531972575, -0.9034285948871803, -1.770059340221131, 1.417516049558281, 1.7792033261567348], a=0.7853981633974483, v=0.7853981633974483)
                else:
                  $ 286 "ElseIf read_port_register(robot_pose_164)≟5"
                  if ( read_port_register (robot_pose_164) == 5):
                    $ 287 "c_p≔get_actual_tcp_pose()"
                    global c_p= get_actual_tcp_pose ()
                    $ 288 "MoveL"
                    $ 289 "m_p≔pose_trans(c_p, p[0,0,0,d2r(tilt_deg_man),0,0])"
                    global m_p= pose_trans (c_p, p[0,0,0,d2r(tilt_deg_man),0,0])
                    $ 290 "m_p" "breakAfter"
                    movel(pose_trans(Base, m_p), a=0.03, v=0.03)
                    $ 291 "m_p≔pose_trans(c_p, p[0,0,0,d2r(-tilt_deg_man),0,0])"
                    global m_p= pose_trans (c_p, p[0,0,0,d2r(-tilt_deg_man),0,0])
                    $ 292 "m_p" "breakAfter"
                    movel(pose_trans(Base, m_p), a=0.03, v=0.03)
                    $ 293 "c_p" "breakAfter"
                    movel(pose_trans(Base, c_p), a=0.03, v=0.03)
                    $ 294 "m_p≔pose_trans(c_p, p[0,0,0,0,d2r(tilt_deg_man),0])"
                    global m_p= pose_trans (c_p, p[0,0,0,0,d2r(tilt_deg_man),0])
                    $ 295 "m_p" "breakAfter"
                    movel(pose_trans(Base, m_p), a=0.03, v=0.03)
                    $ 296 "m_p≔pose_trans(c_p, p[0,0,0,0,d2r(-tilt_deg_man),0])"
                    global m_p= pose_trans (c_p, p[0,0,0,0,d2r(-tilt_deg_man),0])
                    $ 297 "m_p" "breakAfter"
                    movel(pose_trans(Base, m_p), a=0.03, v=0.03)
                    $ 298 "c_p" "breakAfter"
                    movel(pose_trans(Base, c_p), a=0.03, v=0.03)
                    $ 299 "m_p≔pose_trans(c_p, p[0,0,0,0,0,d2r(tilt_deg_man)])"
                    global m_p= pose_trans (c_p, p[0,0,0,0,0,d2r(tilt_deg_man)])
                    $ 300 "m_p" "breakAfter"
                    movel(pose_trans(Base, m_p), a=0.03, v=0.03)
                    $ 301 "m_p≔pose_trans(c_p, p[0,0,0,0,0,d2r(-tilt_deg_man)])"
                    global m_p= pose_trans (c_p, p[0,0,0,0,0,d2r(-tilt_deg_man)])
                    $ 302 "m_p" "breakAfter"
                    movel(pose_trans(Base, m_p), a=0.03, v=0.03)
                    $ 303 "c_p" "breakAfter"
                    movel(pose_trans(Base, c_p), a=0.03, v=0.03)
                  end
                end
              end
            end
          end
          $ 304 "Call Move_done"
          Move_done()
        end
      end
      $ 305 "Call robotand_cell_initalizat"
      robotand_cell_initalizat()
    else:
      $ 306 "ElseIf a0_Job_Mode≟2"
      global thread_flag_306=0
      thread Thread_if_306():
        $ 307 "'JOB_AUTO'"
        # 'JOB_AUTO'
        $ 308 "auto_on≔ True "
        global auto_on=  True
        $ 309 "Init"
        $ 310 "If freedrive_trg"
        if (freedrive_trg):
          $ 311 "end_freedrive_mode()"
          end_freedrive_mode()
          $ 312 "freedrive_trg≔ False "
          global freedrive_trg=  False
        end
        $ 313 "write_port_register(202,0)"
        write_port_register(202,0)
        $ 314 "write_port_register(robot_ready_141,0)"
        write_port_register(robot_ready_141,0)
        $ 315 "homeing()"
        homeing()
        $ 316 "Wait: 0.2"
        sleep(0.2)
        $ 317 "Cell_calculation"
        $ 318 "'setting'"
        # 'setting'
        $ 319 "Auto_trig≔ False "
        global Auto_trig=  False
        $ 320 "If Auto_trig≟ False "
        if (Auto_trig ==   False  ):
          $ 321 "If simulation_mode"
          if (simulation_mode):
            $ 322 "b1_cell_info_L≔B"
            global b1_cell_info_L=B
            $ 323 "b1_cell_info_R≔B"
            global b1_cell_info_R=B
            $ 324 "b1_cell_select≔motion_num([A_VL1,A_VR1,A_HOR,0,0,0])"
            global b1_cell_select=motion_num([A_VL1,A_VR1,A_HOR,0,0,0])
            $ 325 "b1_cell_select≔motion_num([A_HOR,0,0,0,0,0])"
            global b1_cell_select=motion_num([A_HOR,0,0,0,0,0])
            $ 326 "EXT_flag1≔integer_to_binary_list(read_port_register(2048))"
            global EXT_flag1= integer_to_binary_list ( read_port_register (2048))
            $ 327 "b1_cell_thickne≔6"
            global b1_cell_thickne=6
            $ 328 "A_Touch_trig_l≔touch_cal(b1_cell_info_L,b1_cell_info_R,b1_cell_select)"
            global A_Touch_trig_l=touch_cal(b1_cell_info_L,b1_cell_info_R,b1_cell_select)
            $ 329 "Auto_W_num≔cell_motion(A_Touch_trig_l,b1_cell_thickne,EXT_flag1,b1_cell_info_L,b1_cell_info_R)"
            global Auto_W_num=cell_motion(A_Touch_trig_l,b1_cell_thickne,EXT_flag1,b1_cell_info_L,b1_cell_info_R)
            $ 331 "Auto_total_cell≔cell_num(Auto_W_num)"
            global Auto_total_cell=cell_num(Auto_W_num)
            $ 332 "Auto_trig≔ True "
            global Auto_trig=  True
            $ 333 "A_sel_v≔Auto_W_num[0]"
            global A_sel_v=Auto_W_num[0]
          else:
            $ 334 "Else" "noBreak"
            $ 335 "b1_cell_info_L≔read_port_register(171)"
            global b1_cell_info_L= read_port_register (171)
            $ 336 "b1_cell_info_R≔read_port_register(172)"
            global b1_cell_info_R= read_port_register (172)
            $ 337 "EXT_flag1≔integer_to_binary_list(read_port_register(179))"
            global EXT_flag1= integer_to_binary_list ( read_port_register (179))
            $ 338 "b1_cell_select≔read_port_register(178)"
            global b1_cell_select= read_port_register (178)
            $ 339 "b1_cell_thickne≔read_port_register(183)"
            global b1_cell_thickne= read_port_register (183)
            $ 340 "A_Touch_trig_l≔touch_cal(b1_cell_info_L,b1_cell_info_R,b1_cell_select)"
            global A_Touch_trig_l=touch_cal(b1_cell_info_L,b1_cell_info_R,b1_cell_select)
            $ 341 "Auto_W_num≔cell_motion(A_Touch_trig_l,b1_cell_thickne,EXT_flag1,b1_cell_info_L,b1_cell_info_R)"
            global Auto_W_num=cell_motion(A_Touch_trig_l,b1_cell_thickne,EXT_flag1,b1_cell_info_L,b1_cell_info_R)
            $ 342 "Auto_total_cell≔cell_num(Auto_W_num)"
            global Auto_total_cell=cell_num(Auto_W_num)
            $ 343 "Auto_trig≔ True "
            global Auto_trig=  True
            $ 344 "A_sel_v≔Auto_W_num[0]"
            global A_sel_v=Auto_W_num[0]
          end
          $ 345 "write_port_register(139,Auto_total_cell-1)"
          write_port_register(139,Auto_total_cell-1)
        end
        $ 346 "Auto_cur_cell≔0"
        global Auto_cur_cell=0
        $ 347 "Touch,Welding"
        $ 348 "'Calculate total sequence and decide way'"
        # 'Calculate total sequence and decide way'
        $ 349 "Calculate & Move & Touch"
        $ 350 "touch_init"
        $ 351 "Call cell_info"
        cell_info()
        $ 352 "If simulation_mode"
        if (simulation_mode):
          $ 353 "Call welding_parameter_sim"
          welding_parameter_sim()
        else:
          $ 354 "Else" "noBreak"
          $ 355 "Call welding_parameter_init"
          welding_parameter_init()
          $ 356 "touch_temp≔read_port_register(180)"
          global touch_temp= read_port_register (180)
          $ 357 "A_cur_2f≔0"
          global A_cur_2f=0
          $ 358 "wv_direction≔1"
          global wv_direction=1
        end
        $ 359 "If touch_temp≟0"
        if (touch_temp == 0):
          $ 360 "reset Variable"
          $ 361 "A_Prepos_l=[p[0, 0, 0, 0, 0, 0], p[0, 0, 0, 0, 0, 0], p[0, 0, 0, 0, 0, 0],p[0, 0, 0, 0, 0, 0], p[0, 0, 0, 0, 0, 0], p[0, 0, 0, 0, 0, 0], p[0, 0, 0, 0, 0, 0], p[0, 0, 0, 0, 0, 0], p[0, 0, 0, 0, 0, 0], p[0, 0, 0, 0, 0, 0], p[0, 0, 0, 0, 0, 0],p[0, 0, 0, 0, 0, 0],p[0, 0, 0, 0, 0, 0],p[0, 0, 0, 0, 0, 0],p[0, 0, 0, 0, 0, 0],p[0,0,0,0,0,0]]"
          A_Prepos_l=[p[0, 0, 0, 0, 0, 0], p[0, 0, 0, 0, 0, 0], p[0, 0, 0, 0, 0, 0],p[0, 0, 0, 0, 0, 0], p[0, 0, 0, 0, 0, 0], p[0, 0, 0, 0, 0, 0], p[0, 0, 0, 0, 0, 0], p[0, 0, 0, 0, 0, 0], p[0, 0, 0, 0, 0, 0], p[0, 0, 0, 0, 0, 0], p[0, 0, 0, 0, 0, 0],p[0, 0, 0, 0, 0, 0],p[0, 0, 0, 0, 0, 0],p[0, 0, 0, 0, 0, 0],p[0, 0, 0, 0, 0, 0],p[0,0,0,0,0,0]]
          $ 362 "A_Touch_p=[p[0, 0, 0, 0, 0, 0], p[0, 0, 0, 0, 0, 0], p[0, 0, 0, 0, 0, 0],p[0, 0, 0, 0, 0, 0], p[0, 0, 0, 0, 0, 0], p[0, 0, 0, 0, 0, 0], p[0, 0, 0, 0, 0, 0], p[0, 0, 0, 0, 0, 0], p[0, 0, 0, 0, 0, 0], p[0, 0, 0, 0, 0, 0], p[0, 0, 0, 0, 0, 0],p[0, 0, 0, 0, 0, 0],p[0, 0, 0, 0, 0, 0],p[0, 0, 0, 0, 0, 0],p[0, 0, 0, 0, 0, 0],p[0,0,0,0,0,0]]"
          A_Touch_p=[p[0, 0, 0, 0, 0, 0], p[0, 0, 0, 0, 0, 0], p[0, 0, 0, 0, 0, 0],p[0, 0, 0, 0, 0, 0], p[0, 0, 0, 0, 0, 0], p[0, 0, 0, 0, 0, 0], p[0, 0, 0, 0, 0, 0], p[0, 0, 0, 0, 0, 0], p[0, 0, 0, 0, 0, 0], p[0, 0, 0, 0, 0, 0], p[0, 0, 0, 0, 0, 0],p[0, 0, 0, 0, 0, 0],p[0, 0, 0, 0, 0, 0],p[0, 0, 0, 0, 0, 0],p[0, 0, 0, 0, 0, 0],p[0,0,0,0,0,0]]
          $ 363 "reset_par"
          $ 364 "for_cal_rot≔p[0,0,0,0,0,0]"
          global for_cal_rot=p[0,0,0,0,0,0]
          $ 365 "for_cal_zr≔p[0,0,0,0,0,0]"
          global for_cal_zr=p[0,0,0,0,0,0]
          $ 366 "for_z_VLR2≔p[0,0,0,0,0,0]"
          global for_z_VLR2=p[0,0,0,0,0,0]
          $ 367 "for_cal_x_wel≔p[0,0,0,0,0,0]"
          global for_cal_x_wel=p[0,0,0,0,0,0]
          $ 368 "for_cal_xy≔p[0,0,0,0,0,0]"
          global for_cal_xy=p[0,0,0,0,0,0]
          $ 369 "for_cal_y_wel≔p[0,0,0,0,0,0]"
          global for_cal_y_wel=p[0,0,0,0,0,0]
          $ 370 "for_x_HOR≔p[0,0,0,0,0,0]"
          global for_x_HOR=p[0,0,0,0,0,0]
          $ 371 "for_x_HOR_R≔p[0,0,0,0,0,0]"
          global for_x_HOR_R=p[0,0,0,0,0,0]
          $ 372 "for_z_VL1≔p[0,0,0,0,0,0]"
          global for_z_VL1=p[0,0,0,0,0,0]
          $ 373 "for_z_VR1≔p[0,0,0,0,0,0]"
          global for_z_VR1=p[0,0,0,0,0,0]
        end
        $ 374 "write_port_register(143,0)"
        write_port_register(143,0)
        $ 375 "write_port_register(144,0)"
        write_port_register(144,0)
        $ 376 "timer_1: Reset"
        timer_1 = 0
        $ 377 "EXT_flag1≔integer_to_binary_list(read_port_register(179))"
        global EXT_flag1= integer_to_binary_list ( read_port_register (179))
        $ 379 "If touch_temp≟0"
        if (touch_temp == 0):
          $ 380 "write_port_register(138,0)"
          write_port_register(138,0)
          $ 381 "Call reset_multi_record"
          reset_multi_record()
          $ 382 "get_touch_position"
          $ 383 "get pre-positions"
          $ 384 "If read_port_register(work_type_165)≟2"
          if ( read_port_register (work_type_165) == 2):
            $ 385 "freedrive touch"
            $ 386 "move_i≔1"
            global move_i=1
            $ 387 "Loop move_i<9"
            while (move_i<9):
              $ 388 "Wait: 0.1"
              sleep(0.1)
              $ 389 "Wait save_tool=LO"
              while (get_tool_digital_in(0) == True):
                sync()
              end
              $ 390 "If A_Touch_trig_l[move_i]≟ True "
              if (A_Touch_trig_l[move_i] ==   True  ):
                $ 391 "If move_i≟A_HOR"
                if (move_i == A_HOR):
                  $ 392 "If b1_cell_info_L≟B or b1_cell_info_L≟D or b1_cell_info_L≟d or A_Prepos_l[A_VL1]≟p[0,0,0,0,0,0]"
                  if (b1_cell_info_L == B  or  b1_cell_info_L == D  or  b1_cell_info_L == d  or  A_Prepos_l[A_VL1] == p[0,0,0,0,0,0]):
                    $ 393 "write_port_register(touch_cell_155,5)"
                    write_port_register(touch_cell_155,5)
                    $ 394 "write_port_register(touch_num_156,1)"
                    write_port_register(touch_num_156,1)
                    $ 395 "Call touch_sub"
                    touch_sub()
                    $ 396 "g_cp≔get_actual_tcp_pose()"
                    global g_cp= get_actual_tcp_pose ()
                    $ 397 "If g_cp[2]<(get_margin_z+a7_cell_bottom)/1000"
                    if (g_cp[2]<(get_margin_z+a7_cell_bottom)/1000):
                      $ 398 "g_cp[2]=(get_margin_z+a7_cell_bottom)/1000"
                      g_cp[2]=(get_margin_z+a7_cell_bottom)/1000
                    end
                    $ 399 "A_Prepos_l[move_i]=g_cp"
                    A_Prepos_l[move_i]=g_cp
                  end
                else:
                  $ 400 "ElseIf move_i≟A_HOR_ML"
                  if (move_i == A_HOR_ML):
                    $ 401 "If b1_cell_info_L≟B or b1_cell_info_L≟D or b1_cell_info_L≟d or A_Prepos_l[A_VL1]≟p[0,0,0,0,0,0]"
                    if (b1_cell_info_L == B  or  b1_cell_info_L == D  or  b1_cell_info_L == d  or  A_Prepos_l[A_VL1] == p[0,0,0,0,0,0]):
                      $ 402 "write_port_register(touch_cell_155,5)"
                      write_port_register(touch_cell_155,5)
                      $ 403 "write_port_register(touch_num_156,3)"
                      write_port_register(touch_num_156,3)
                      $ 404 "Call touch_sub"
                      touch_sub()
                      $ 405 "g_cp≔get_actual_tcp_pose()"
                      global g_cp= get_actual_tcp_pose ()
                      $ 406 "If g_cp[2]<(get_margin_z+a7_cell_bottom)/1000"
                      if (g_cp[2]<(get_margin_z+a7_cell_bottom)/1000):
                        $ 407 "g_cp[2]=(get_margin_z+a7_cell_bottom)/1000"
                        g_cp[2]=(get_margin_z+a7_cell_bottom)/1000
                      end
                      $ 408 "A_Prepos_l[move_i]=g_cp"
                      A_Prepos_l[move_i]=g_cp
                    end
                  else:
                    $ 409 "ElseIf move_i≟A_HOR_R"
                    if (move_i == A_HOR_R):
                      $ 410 "If b1_cell_info_L≟B or b1_cell_info_L≟D or b1_cell_info_L≟d or A_Prepos_l[A_VL1]≟p[0,0,0,0,0,0]"
                      if (b1_cell_info_L == B  or  b1_cell_info_L == D  or  b1_cell_info_L == d  or  A_Prepos_l[A_VL1] == p[0,0,0,0,0,0]):
                        $ 411 "write_port_register(touch_cell_155,5)"
                        write_port_register(touch_cell_155,5)
                        $ 412 "write_port_register(touch_num_156,2)"
                        write_port_register(touch_num_156,2)
                        $ 413 "Call touch_sub"
                        touch_sub()
                        $ 414 "g_cp≔get_actual_tcp_pose()"
                        global g_cp= get_actual_tcp_pose ()
                        $ 415 "If g_cp[2]<(get_margin_z+a7_cell_bottom)/1000"
                        if (g_cp[2]<(get_margin_z+a7_cell_bottom)/1000):
                          $ 416 "g_cp[2]=(get_margin_z+a7_cell_bottom)/1000"
                          g_cp[2]=(get_margin_z+a7_cell_bottom)/1000
                        end
                        $ 417 "A_Prepos_l[move_i]=g_cp"
                        A_Prepos_l[move_i]=g_cp
                      end
                    else:
                      $ 418 "ElseIf move_i≟A_HOR_MR"
                      if (move_i == A_HOR_MR):
                        $ 419 "If b1_cell_info_L≟B or b1_cell_info_L≟D or b1_cell_info_L≟d or A_Prepos_l[A_VL1]≟p[0,0,0,0,0,0]"
                        if (b1_cell_info_L == B  or  b1_cell_info_L == D  or  b1_cell_info_L == d  or  A_Prepos_l[A_VL1] == p[0,0,0,0,0,0]):
                          $ 420 "write_port_register(touch_cell_155,5)"
                          write_port_register(touch_cell_155,5)
                          $ 421 "write_port_register(touch_num_156,4)"
                          write_port_register(touch_num_156,4)
                          $ 422 "Call touch_sub"
                          touch_sub()
                          $ 423 "g_cp≔get_actual_tcp_pose()"
                          global g_cp= get_actual_tcp_pose ()
                          $ 424 "If g_cp[2]<(get_margin_z+a7_cell_bottom)/1000"
                          if (g_cp[2]<(get_margin_z+a7_cell_bottom)/1000):
                            $ 425 "g_cp[2]=(get_margin_z+a7_cell_bottom)/1000"
                            g_cp[2]=(get_margin_z+a7_cell_bottom)/1000
                          end
                          $ 426 "A_Prepos_l[move_i]=g_cp"
                          A_Prepos_l[move_i]=g_cp
                        end
                      else:
                        $ 427 "Else" "noBreak"
                        $ 428 "write_port_register(touch_cell_155,move_i)"
                        write_port_register(touch_cell_155,move_i)
                        $ 429 "write_port_register(touch_num_156,1)"
                        write_port_register(touch_num_156,1)
                        $ 430 "Call touch_sub"
                        touch_sub()
                        $ 431 "A_Prepos_l[move_i]=get_actual_tcp_pose()"
                        A_Prepos_l[move_i]= get_actual_tcp_pose ()
                        $ 432 "If move_i≤4"
                        if (move_i <= 4):
                          $ 433 "write_port_register(touch_cell_155,move_i)"
                          write_port_register(touch_cell_155,move_i)
                          $ 434 "write_port_register(touch_num_156,2)"
                          write_port_register(touch_num_156,2)
                          $ 435 "Wait: 0.1"
                          sleep(0.1)
                          $ 436 "Call touch_sub"
                          touch_sub()
                          $ 437 "A_Prepos_l[move_i+9]=get_actual_tcp_pose()"
                          A_Prepos_l[move_i+9]= get_actual_tcp_pose ()
                        end
                      end
                    end
                  end
                end
              else:
                $ 438 "Else" "noBreak"
                $ 439 "A_Prepos_l[move_i]=p[0,0,0,0,0,0]"
                A_Prepos_l[move_i]=p[0,0,0,0,0,0]
                $ 440 "If move_i≤4"
                if (move_i <= 4):
                  $ 441 "A_Prepos_l[move_i+7]=p[0,0,0,0,0,0]"
                  A_Prepos_l[move_i+7]=p[0,0,0,0,0,0]
                else:
                  $ 442 "ElseIf move_i≟A_HOR"
                  if (move_i == A_HOR):
                    $ 443 "A_Prepos_l[A_HOR_ML]=p[0,0,0,0,0,0]"
                    A_Prepos_l[A_HOR_ML]=p[0,0,0,0,0,0]
                    $ 444 "A_Prepos_l[A_HOR_MR]=p[0,0,0,0,0,0]"
                    A_Prepos_l[A_HOR_MR]=p[0,0,0,0,0,0]
                    $ 445 "A_Prepos_l[A_HOR_M]=p[0,0,0,0,0,0]"
                    A_Prepos_l[A_HOR_M]=p[0,0,0,0,0,0]
                    $ 446 "A_Prepos_l[A_HOR_R]=p[0,0,0,0,0,0]"
                    A_Prepos_l[A_HOR_R]=p[0,0,0,0,0,0]
                  end
                end
              end
              $ 447 "move_i≔move_i+1"
              global move_i=move_i+1
            end
            $ 448 "change deg"
            $ 449 "move_i≔1"
            global move_i=1
            $ 450 "Loop move_i<14"
            while (move_i<14):
              $ 451 "If A_Prepos_l[move_i]≠p[0,0,0,0,0,0]"
              if (A_Prepos_l[move_i] != p[0,0,0,0,0,0]):
                $ 452 "If move_i≟A_VL1 or move_i≟A_VL2 or move_i≟A_VL1_END or move_i≟A_VL2_END"
                if (move_i == A_VL1  or  move_i == A_VL2  or  move_i == A_VL1_END  or  move_i == A_VL2_END):
                  $ 453 "b2_left_par≔ True "
                  global b2_left_par=  True
                  $ 454 "b8_wv_2f≔ False "
                  global b8_wv_2f=  False
                  $ 455 "get_pos≔A_Prepos_l[move_i]"
                  global get_pos=A_Prepos_l[move_i]
                  $ 456 "get_org≔left"
                  global get_org=p[.480496318984, .411279115151, .006998291210, -2.211681476386, -.899147924387, -1.383032568605]
                  $ 457 "get_pos≔p[get_pos[0],get_pos[1],get_pos[2],get_org[3],get_org[4],get_org[5]]"
                  global get_pos=p[get_pos[0],get_pos[1],get_pos[2],get_org[3],get_org[4],get_org[5]]
                  $ 458 "pre_tp≔tilt_3f_fun(get_pos,[0,0],a5_f_hole[1])"
                  global pre_tp=tilt_3f_fun(get_pos,[0,0],a5_f_hole[1])
                else:
                  $ 459 "ElseIf move_i≟A_VR1 or move_i≟A_VR2 or move_i≟A_VR1_END or move_i≟A_VR2_END"
                  if (move_i == A_VR1  or  move_i == A_VR2  or  move_i == A_VR1_END  or  move_i == A_VR2_END):
                    $ 460 "b2_left_par≔ False "
                    global b2_left_par=  False
                    $ 461 "b8_wv_2f≔ False "
                    global b8_wv_2f=  False
                    $ 462 "get_pos≔A_Prepos_l[move_i]"
                    global get_pos=A_Prepos_l[move_i]
                    $ 463 "get_org≔right"
                    global get_org=p[.475000000000, -.421403215678, .026417194146, 1.917761036827, -1.141682393512, 1.523356199292]
                    $ 464 "get_pos≔p[get_pos[0],get_pos[1],get_pos[2],get_org[3],get_org[4],get_org[5]]"
                    global get_pos=p[get_pos[0],get_pos[1],get_pos[2],get_org[3],get_org[4],get_org[5]]
                    $ 465 "pre_tp≔tilt_3f_fun(get_pos,[0,0],a5_f_hole[1])"
                    global pre_tp=tilt_3f_fun(get_pos,[0,0],a5_f_hole[1])
                  else:
                    $ 466 "ElseIf move_i≟A_HOR or move_i≟A_HOR_ML"
                    if (move_i == A_HOR  or  move_i == A_HOR_ML):
                      $ 467 "b8_wv_2f≔ True "
                      global b8_wv_2f=  True
                      $ 468 "b2_left_par≔ True "
                      global b2_left_par=  True
                      $ 469 "get_pos≔A_Prepos_l[move_i]"
                      global get_pos=A_Prepos_l[move_i]
                      $ 470 "get_org≔up_left"
                      global get_org=p[.492775857339, .409517380626, -.029063830209, -2.419264859926, -.998084331190, -1.368689080860]
                      $ 471 "get_pos≔p[get_pos[0],get_pos[1],get_pos[2],get_org[3],get_org[4],get_org[5]]"
                      global get_pos=p[get_pos[0],get_pos[1],get_pos[2],get_org[3],get_org[4],get_org[5]]
                      $ 472 "pre_tp≔tilt_2f_fun(get_pos,[0,0], True , True )"
                      global pre_tp=tilt_2f_fun(get_pos,[0,0],  True  ,  True  )
                    else:
                      $ 473 "ElseIf move_i≟A_HOR_R or move_i≟A_HOR_MR"
                      if (move_i == A_HOR_R  or  move_i == A_HOR_MR):
                        $ 474 "b8_wv_2f≔ True "
                        global b8_wv_2f=  True
                        $ 475 "b2_left_par≔ False "
                        global b2_left_par=  False
                        $ 476 "get_pos≔A_Prepos_l[move_i]"
                        global get_pos=A_Prepos_l[move_i]
                        $ 477 "get_org≔up_right"
                        global get_org=p[.445203173045, -.406687378356, -.031125942276, 2.308490741423, -1.066468937023, 1.322151316133]
                        $ 478 "get_pos≔p[get_pos[0],get_pos[1],get_pos[2],get_org[3],get_org[4],get_org[5]]"
                        global get_pos=p[get_pos[0],get_pos[1],get_pos[2],get_org[3],get_org[4],get_org[5]]
                        $ 479 "pre_tp≔tilt_2f_fun(get_pos,[0,0], False , True )"
                        global pre_tp=tilt_2f_fun(get_pos,[0,0],  False  ,  True  )
                      end
                    end
                  end
                end
                $ 480 "A_Prepos_l[move_i]=pre_tp"
                A_Prepos_l[move_i]=pre_tp
              end
              $ 481 "move_i≔move_i+1"
              global move_i=move_i+1
            end
            $ 482 "homeing()"
            homeing()
            $ 483 "Wait read_port_register(170)≟1"
            while (not( read_port_register (170) == 1)):
              sync()
            end
            $ 484 "write_port_register(170,0)"
            write_port_register(170,0)
          else:
            $ 485 "Else" "noBreak"
            $ 486 "value from pendant"
            $ 487 "move_i≔1"
            global move_i=1
            $ 489 "Touch_FrontandSide"
            $ 490 "If EXT_flag1[11]≟ True "
            if (EXT_flag1[11] ==   True  ):
              $ 491 "Touch front and side_Right"
              $ 492 "move_center≔pose_add(first_p_wp, p[-first_p_wp[0]+(get_center-work_touch_dis)/1000,0,0,0,0,0])"
              global move_center= pose_add (first_p_wp, p[-first_p_wp[0]+(get_center-work_touch_dis)/1000,0,0,0,0,0])
              $ 493 "get_pose_side_t≔0"
              global get_pose_side_t=0
              $ 495 "move_center[2]=(center_height+a7_cell_bottom)/1000"
              move_center[2]=(center_height+a7_cell_bottom)/1000
              $ 497 "MoveL"
              $ 498 "move_center" "breakAfter"
              movel(pose_trans(Base, move_center), a=0.5, v=0.15)
              $ 499 "touch_center≔contact_fun(p[0,0,0,0,0,0],[1,0,0],20000,20,20)"
              global touch_center=contact_fun(p[0,0,0,0,0,0],[1,0,0],20000,20,20)
              $ 500 "direction(p[0,0,0,0,0,0],[-1,0,0],10,180,200)"
              direction(p[0,0,0,0,0,0],[-1,0,0],10,180,200)
              $ 501 "get_center≔touch_center[0]*1000"
              global get_center=touch_center[0]*1000
              $ 502 "a7_f_distance≔get_center"
              global a7_f_distance=get_center
              $ 503 "move_center≔pose_add(move_center,p[0,sec_touch_dis/1000,0,0,0,0])"
              global move_center= pose_add (move_center,p[0,sec_touch_dis/1000,0,0,0,0])
              $ 504 "move_center[0]=touch_center[0]-20/1000"
              move_center[0]=touch_center[0]-20/1000
              $ 505 "MoveL"
              $ 506 "move_center" "breakAfter"
              movel(pose_trans(Base, move_center), a=0.5, v=0.15)
              $ 507 "touch_center2≔contact_fun(p[0,0,0,0,0,0],[1,0,0],20000,20,20)"
              global touch_center2=contact_fun(p[0,0,0,0,0,0],[1,0,0],20000,20,20)
              $ 508 "center_line≔get_feature_Line(touch_center,touch_center2)"
              global center_line=get_feature_Line(touch_center,touch_center2)
              $ 509 "direction(p[0,0,0,0,0,0],[-1,0,0],10,180,200)"
              direction(p[0,0,0,0,0,0],[-1,0,0],10,180,200)
              $ 510 "g_current_p≔get_actual_tcp_pose()"
              global g_current_p= get_actual_tcp_pose ()
              $ 511 "g_current_p≔pose_trans(g_current_p, p[0,0,0,0,d2r(-3),0])"
              global g_current_p= pose_trans (g_current_p, p[0,0,0,0,d2r(-3),0])
              $ 512 "MoveL"
              $ 513 "g_current_p" "breakAfter"
              movel(pose_trans(Base, g_current_p), a=0.1, v=0.05)
              $ 514 "A_touch_bottom≔contact_fun(p[0,0,0,0,0,0],[0,0,-1],20000,20,20)"
              global A_touch_bottom=contact_fun(p[0,0,0,0,0,0],[0,0,-1],20000,20,20)
              $ 515 "direction(p[0,0,0,0,0,0],[0,0,1],15,180,200)"
              direction(p[0,0,0,0,0,0],[0,0,1],15,180,200)
              $ 517 "homeing()"
              homeing()
              $ 518 "b2_left_par≔ False "
              global b2_left_par=  False
              $ 519 "b8_wv_2f≔ False "
              global b8_wv_2f=  False
              $ 520 "b2_cell≔b1_cell_info_R"
              global b2_cell=b1_cell_info_R
              $ 521 "touch_side≔p[0,(-a6_f_width/2)/1000,0,0,0,0]"
              global touch_side=p[0,(-a6_f_width/2)/1000,0,0,0,0]
              $ 522 "get_pos≔get_lr(side_p_R,a6_f_width,[35,0,0,0,0],a7_f_distance-20,b2_left_par,b8_wv_2f,Touch_dis,get_margin_z,touch_side,30,0,center_line, True )"
              global get_pos=get_lr(p[.471584857321, -.427242166643, .026448165242, 1.806736638758, -1.227818761912, 1.383474453522],a6_f_width,[35,0,0,0,0],a7_f_distance-20,b2_left_par,b8_wv_2f,Touch_dis,get_margin_z,touch_side,30,0,center_line,  True  )
              $ 524 "pre_tp≔get_pos"
              global pre_tp=get_pos
              $ 525 "pre_tp≔pose_add(pre_tp, p[side_pos_x/1000,0,0,0,0,0])"
              global pre_tp= pose_add (pre_tp, p[side_pos_x/1000,0,0,0,0,0])
              $ 526 "pre_tp[2]=(center_height+a7_cell_bottom)/1000"
              pre_tp[2]=(center_height+a7_cell_bottom)/1000
              $ 527 "MoveL"
              $ 528 "pre_tp" "breakAfter"
              movel(pose_trans(Base, pre_tp), a=0.8, v=0.4)
              $ 529 "touch_side≔contact_fun(p[0,0,0,0,0,0],[0,-1,0],20000,13,13)"
              global touch_side=contact_fun(p[0,0,0,0,0,0],[0,-1,0],20000,13,13)
              $ 530 "event_cal_on≔ True "
              global event_cal_on=  True
              $ 531 "touch_side≔get_feature_pose(touch_side,center_line)"
              global touch_side=get_feature_pose(touch_side,center_line)
              $ 532 "direction(p[0,0,0,0,0,0],[0,1,0],10,180,200)"
              direction(p[0,0,0,0,0,0],[0,1,0],10,180,200)
              $ 533 "write_welder(4, False )"
              write_welder(4,  False  )
              $ 534 "get_pose_side_t≔touch_side[1]*1000"
              global get_pose_side_t=touch_side[1]*1000
              $ 535 "get_pose_side_t≔get_pose_side_t+(a6_f_width/2)"
              global get_pose_side_t=get_pose_side_t+(a6_f_width/2)
              $ 536 "event_side_on≔ True "
              global event_side_on=  True
              $ 537 "MoveL"
              $ 538 "Direction: Base"
              global move_thread_flag_538=0
              thread move_thread_538():
                enter_critical
                move_thread_flag_538 = 1
                local towardsPos=calculate_point_to_move_towards(p[0.0,0.0,0.0,0.0,0.0,0.0], [-1,1,0], 0.03)
                movel(towardsPos, a=0.3, v=0.15)
                move_thread_flag_538 = 2
                exit_critical
              end
              move_thread_flag_538 = 0
              move_thread_han_538 = run move_thread_538()
              while (True):
                sleep(1.0E-10)
                if (move_thread_flag_538 > 1):
                  join move_thread_han_538
                  $ 539 "Until (distance)"
                  break
                end
                sync()
              end
              $ 540 "homeing()"
              homeing()
            else:
              $ 541 "Else" "noBreak"
              $ 542 "Touch front and side_Left"
              $ 543 "move_center≔pose_add(first_p_wp, p[-first_p_wp[0]+(get_center-work_touch_dis)/1000,0,0,0,0,0])"
              global move_center= pose_add (first_p_wp, p[-first_p_wp[0]+(get_center-work_touch_dis)/1000,0,0,0,0,0])
              $ 544 "get_pose_side_t≔0"
              global get_pose_side_t=0
              $ 546 "move_center[2]=(center_height+a7_cell_bottom)/1000"
              move_center[2]=(center_height+a7_cell_bottom)/1000
              $ 548 "MoveL"
              $ 549 "move_center" "breakAfter"
              movel(pose_trans(Base, move_center), a=0.5, v=0.15)
              $ 550 "touch_center≔contact_fun(p[0,0,0,0,0,0],[1,0,0],20000,20,20)"
              global touch_center=contact_fun(p[0,0,0,0,0,0],[1,0,0],20000,20,20)
              $ 551 "direction(p[0,0,0,0,0,0],[-1,0,0],10,180,200)"
              direction(p[0,0,0,0,0,0],[-1,0,0],10,180,200)
              $ 552 "get_center≔touch_center[0]*1000"
              global get_center=touch_center[0]*1000
              $ 553 "a7_f_distance≔get_center"
              global a7_f_distance=get_center
              $ 554 "move_center≔pose_add(move_center,p[0,sec_touch_dis/1000,0,0,0,0])"
              global move_center= pose_add (move_center,p[0,sec_touch_dis/1000,0,0,0,0])
              $ 555 "move_center[0]=touch_center[0]-20/1000"
              move_center[0]=touch_center[0]-20/1000
              $ 556 "MoveL"
              $ 557 "move_center" "breakAfter"
              movel(pose_trans(Base, move_center), a=0.5, v=0.15)
              $ 558 "touch_center2≔contact_fun(p[0,0,0,0,0,0],[1,0,0],20000,20,20)"
              global touch_center2=contact_fun(p[0,0,0,0,0,0],[1,0,0],20000,20,20)
              $ 559 "center_line≔get_feature_Line(touch_center,touch_center2)"
              global center_line=get_feature_Line(touch_center,touch_center2)
              $ 560 "direction(p[0,0,0,0,0,0],[-1,0,0],10,180,200)"
              direction(p[0,0,0,0,0,0],[-1,0,0],10,180,200)
              $ 561 "g_current_p≔get_actual_tcp_pose()"
              global g_current_p= get_actual_tcp_pose ()
              $ 562 "g_current_p≔pose_trans(g_current_p, p[0,0,0,0,d2r(-3),0])"
              global g_current_p= pose_trans (g_current_p, p[0,0,0,0,d2r(-3),0])
              $ 563 "MoveL"
              $ 564 "g_current_p" "breakAfter"
              movel(pose_trans(Base, g_current_p), a=0.1, v=0.05)
              $ 565 "A_touch_bottom≔contact_fun(p[0,0,0,0,0,0],[0,0,-1],20000,20,20)"
              global A_touch_bottom=contact_fun(p[0,0,0,0,0,0],[0,0,-1],20000,20,20)
              $ 566 "direction(p[0,0,0,0,0,0],[0,0,1],15,180,200)"
              direction(p[0,0,0,0,0,0],[0,0,1],15,180,200)
              $ 568 "homeing()"
              homeing()
              $ 569 "b2_left_par≔ True "
              global b2_left_par=  True
              $ 570 "b8_wv_2f≔ False "
              global b8_wv_2f=  False
              $ 571 "b2_cell≔b1_cell_info_L"
              global b2_cell=b1_cell_info_L
              $ 572 "touch_side≔p[0,(a6_f_width/2)/1000,0,0,0,0]"
              global touch_side=p[0,(a6_f_width/2)/1000,0,0,0,0]
              $ 573 "get_pos≔get_lr(side_p_L,a6_f_width,[35,0,0,0,0],a7_f_distance-20,b2_left_par,b8_wv_2f,Touch_dis,get_margin_z,touch_side,30,0,center_line, True )"
              global get_pos=get_lr(p[.411215372122, .375785944375, -.010176539343, -1.953488355698, -1.125710367676, -1.228829273458],a6_f_width,[35,0,0,0,0],a7_f_distance-20,b2_left_par,b8_wv_2f,Touch_dis,get_margin_z,touch_side,30,0,center_line,  True  )
              $ 575 "pre_tp≔get_pos"
              global pre_tp=get_pos
              $ 576 "pre_tp≔pose_add(pre_tp, p[side_pos_x/1000,0,0,0,0,0])"
              global pre_tp= pose_add (pre_tp, p[side_pos_x/1000,0,0,0,0,0])
              $ 577 "pre_tp[2]=(center_height+a7_cell_bottom)/1000"
              pre_tp[2]=(center_height+a7_cell_bottom)/1000
              $ 578 "MoveL"
              $ 579 "pre_tp" "breakAfter"
              movel(pose_trans(Base, pre_tp), a=0.8, v=0.4)
              $ 580 "touch_side≔contact_fun(p[0,0,0,0,0,0],[0,1,0],20000,13,13)"
              global touch_side=contact_fun(p[0,0,0,0,0,0],[0,1,0],20000,13,13)
              $ 581 "event_cal_on≔ True "
              global event_cal_on=  True
              $ 582 "touch_side≔get_feature_pose(touch_side,center_line)"
              global touch_side=get_feature_pose(touch_side,center_line)
              $ 583 "direction(p[0,0,0,0,0,0],[0,-1,0],10,180,200)"
              direction(p[0,0,0,0,0,0],[0,-1,0],10,180,200)
              $ 584 "write_welder(4, False )"
              write_welder(4,  False  )
              $ 585 "get_pose_side_t≔touch_side[1]*1000"
              global get_pose_side_t=touch_side[1]*1000
              $ 586 "get_pose_side_t≔get_pose_side_t-(a6_f_width/2)"
              global get_pose_side_t=get_pose_side_t-(a6_f_width/2)
              $ 587 "event_side_on≔ True "
              global event_side_on=  True
              $ 588 "MoveL"
              $ 589 "Direction: Base"
              global move_thread_flag_589=0
              thread move_thread_589():
                enter_critical
                move_thread_flag_589 = 1
                local towardsPos=calculate_point_to_move_towards(p[0.0,0.0,0.0,0.0,0.0,0.0], [-1,-1,0], 0.03)
                movel(towardsPos, a=0.3, v=0.15)
                move_thread_flag_589 = 2
                exit_critical
              end
              move_thread_flag_589 = 0
              move_thread_han_589 = run move_thread_589()
              while (True):
                sleep(1.0E-10)
                if (move_thread_flag_589 > 1):
                  join move_thread_han_589
                  $ 590 "Until (distance)"
                  break
                end
                sync()
              end
              $ 591 "homeing()"
              homeing()
            end
            $ 593 "Wait event_cal_on≟ False "
            while (not(event_cal_on ==   False  )):
              sync()
            end
          end
          $ 595 "move and touch"
          $ 596 "Touch Move"
          $ 597 "HOR_L"
          $ 598 "If A_Prepos_l[A_HOR]≠p[0,0,0,0,0,0]"
          if (A_Prepos_l[A_HOR] != p[0,0,0,0,0,0]):
            $ 599 "b2_left_par≔ True "
            global b2_left_par=  True
            $ 600 "b8_wv_2f≔ True "
            global b8_wv_2f=  True
            $ 601 "b7_tilt_degree≔[0,0,0]"
            global b7_tilt_degree=[0,0,0]
            $ 602 "A_sel_v≔A_HOR"
            global A_sel_v=A_HOR
            $ 603 "wv_direction≔1"
            global wv_direction=1
            $ 604 "Call MoveandTouchFun_2f"
            MoveandTouchFun_2f()
            $ 605 "If b1_cell_info_L≟A or b1_cell_info_L≟C or b1_cell_info_L≟c"
            if (b1_cell_info_L == A  or  b1_cell_info_L == C  or  b1_cell_info_L == c):
              $ 606 "If A_Prepos_l[A_VL1]≟p[0,0,0,0,0,0]"
              if (A_Prepos_l[A_VL1] == p[0,0,0,0,0,0]):
                $ 608 "g_tp≔A_Prepos_l[A_HOR]"
                global g_tp=A_Prepos_l[A_HOR]
                $ 611 "Folder"
                $ 612 "g_cp≔get_actual_tcp_pose()"
                global g_cp= get_actual_tcp_pose ()
                $ 613 "g_cp≔pose_trans(g_cp, p[0,0,0,d2r(12),d2r(5),0])"
                global g_cp= pose_trans (g_cp, p[0,0,0,d2r(12),d2r(5),0])
                $ 614 "MoveL"
                $ 615 "g_cp" "breakAfter"
                movel(pose_trans(Base, g_cp), a=0.08, v=0.08)
                $ 616 "for_x_HOR≔contact_fun(A_Touch_p[A_sel_v],[-1*wv_direction,0,0],10000,15,15,  False)"
                global for_x_HOR=contact_fun(A_Touch_p[A_sel_v],[-1*wv_direction,0,0],10000,15,15,  False)
                $ 617 "direction(p[0,0,0,0,0,0],[0,-1,0],20,120,160)"
                direction(p[0,0,0,0,0,0],[0,-1,0],20,120,160)
                $ 618 "write_welder(4, False )"
                write_welder(4,  False  )
              else:
                $ 619 "Else" "noBreak"
                $ 620 "for_x_HOR≔p[0,0,0,0,0,0]"
                global for_x_HOR=p[0,0,0,0,0,0]
              end
            end
            $ 628 "If point_dist(A_Prepos_l[A_HOR], A_Prepos_l[A_VL1])>0.032"
            if (point_dist(A_Prepos_l[A_HOR], A_Prepos_l[A_VL1])>0.032):
              $ 629 "homeing()"
              homeing()
            end
          end
          $ 630 "VL1"
          $ 631 "If A_Prepos_l[A_VL1]≠p[0,0,0,0,0,0]"
          if (A_Prepos_l[A_VL1] != p[0,0,0,0,0,0]):
            $ 632 "b2_left_par≔ True "
            global b2_left_par=  True
            $ 633 "b8_wv_2f≔ False "
            global b8_wv_2f=  False
            $ 634 "b7_tilt_degree≔[0,0,0]"
            global b7_tilt_degree=[0,0,0]
